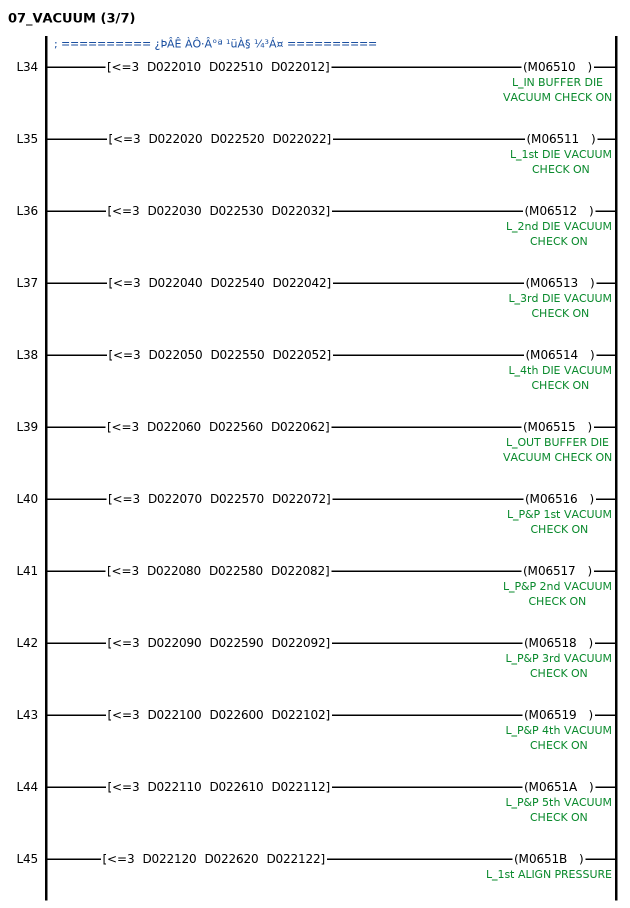
[picture p48: 07_VACUUM rungs L34-L45]
// ========== ¿ÞÂÊ ÀÔ·Â°ª ¹üÀ§ ¼³Á¤ ==========
; L34
LOAD<=3   D022010 D022510 D022012
OUT       M06510	// L_IN BUFFER DIE VACUUM CHECK ON
; L35
LOAD<=3   D022020 D022520 D022022
OUT       M06511	// L_1st DIE VACUUM CHECK ON
; L36
LOAD<=3   D022030 D022530 D022032
OUT       M06512	// L_2nd DIE VACUUM CHECK ON
; L37
LOAD<=3   D022040 D022540 D022042
OUT       M06513	// L_3rd DIE VACUUM CHECK ON
; L38
LOAD<=3   D022050 D022550 D022052
OUT       M06514	// L_4th DIE VACUUM CHECK ON
; L39
LOAD<=3   D022060 D022560 D022062
OUT       M06515	// L_OUT BUFFER DIE VACUUM CHECK ON
; L40
LOAD<=3   D022070 D022570 D022072
OUT       M06516	// L_P&P 1st VACUUM CHECK ON
; L41
LOAD<=3   D022080 D022580 D022082
OUT       M06517	// L_P&P 2nd VACUUM CHECK ON
; L42
LOAD<=3   D022090 D022590 D022092
OUT       M06518	// L_P&P 3rd VACUUM CHECK ON
; L43
LOAD<=3   D022100 D022600 D022102
OUT       M06519	// L_P&P 4th VACUUM CHECK ON
; L44
LOAD<=3   D022110 D022610 D022112
OUT       M0651A	// L_P&P 5th VACUUM CHECK ON
; L45
LOAD<=3   D022120 D022620 D022122
OUT       M0651B	// L_1st ALIGN PRESSURE

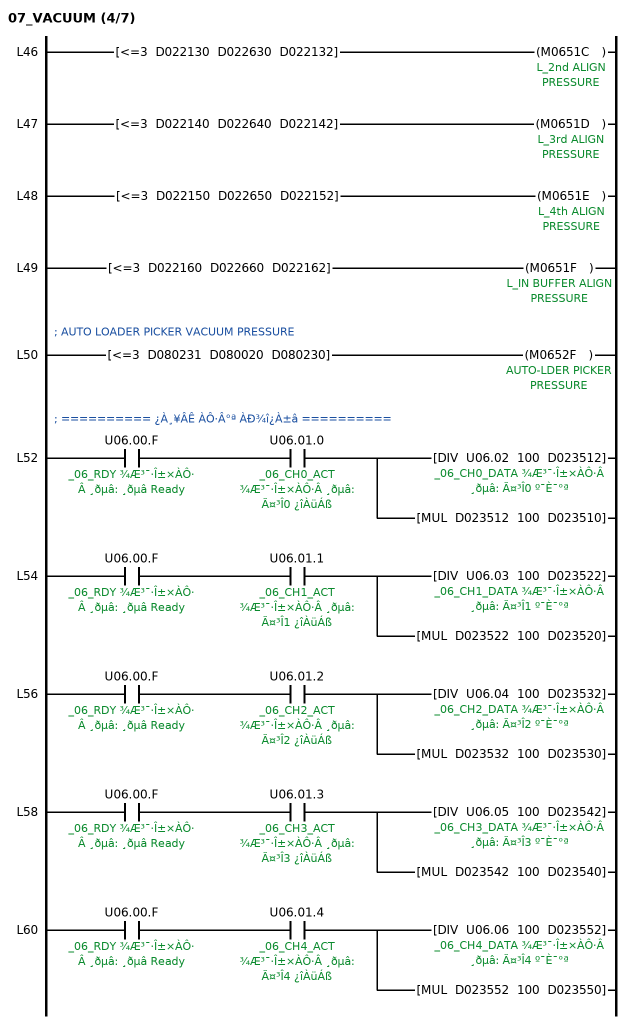
; L46
LOAD<=3   D022130 D022630 D022132
OUT       M0651C	// L_2nd ALIGN PRESSURE
; L47
LOAD<=3   D022140 D022640 D022142
OUT       M0651D	// L_3rd ALIGN PRESSURE
; L48
LOAD<=3   D022150 D022650 D022152
OUT       M0651E	// L_4th ALIGN PRESSURE
; L49
LOAD<=3   D022160 D022660 D022162
OUT       M0651F	// L_IN BUFFER ALIGN PRESSURE
; L50
LOAD<=3   D080231 D080020 D080230
OUT       M0652F	// AUTO-LDER PICKER PRESSURE
// output comment: AUTO LOADER PICKER VACUUM PRESSURE
// ========== ¿À¸¥ÂÊ ÀÔ·Â°ª ÀÐ¾î¿À±â ==========
; L52
LOAD      U06.00.F	// _06_RDY ¾Æ³¯·Î±×ÀÔ·Â ¸ðµâ: ¸ðµâ Ready
AND       U06.01.0	// _06_CH0_ACT ¾Æ³¯·Î±×ÀÔ·Â ¸ðµâ: Ã¤³Î0 ¿îÀüÁß
DIV       U06.02 100 D023512	// _06_CH0_DATA ¾Æ³¯·Î±×ÀÔ·Â ¸ðµâ: Ã¤³Î0 º¯È¯°ª
MUL       D023512 100 D023510
; L54
LOAD      U06.00.F	// _06_RDY ¾Æ³¯·Î±×ÀÔ·Â ¸ðµâ: ¸ðµâ Ready
AND       U06.01.1	// _06_CH1_ACT ¾Æ³¯·Î±×ÀÔ·Â ¸ðµâ: Ã¤³Î1 ¿îÀüÁß
DIV       U06.03 100 D023522	// _06_CH1_DATA ¾Æ³¯·Î±×ÀÔ·Â ¸ðµâ: Ã¤³Î1 º¯È¯°ª
MUL       D023522 100 D023520
; L56
LOAD      U06.00.F	// _06_RDY ¾Æ³¯·Î±×ÀÔ·Â ¸ðµâ: ¸ðµâ Ready
AND       U06.01.2	// _06_CH2_ACT ¾Æ³¯·Î±×ÀÔ·Â ¸ðµâ: Ã¤³Î2 ¿îÀüÁß
DIV       U06.04 100 D023532	// _06_CH2_DATA ¾Æ³¯·Î±×ÀÔ·Â ¸ðµâ: Ã¤³Î2 º¯È¯°ª
MUL       D023532 100 D023530
; L58
LOAD      U06.00.F	// _06_RDY ¾Æ³¯·Î±×ÀÔ·Â ¸ðµâ: ¸ðµâ Ready
AND       U06.01.3	// _06_CH3_ACT ¾Æ³¯·Î±×ÀÔ·Â ¸ðµâ: Ã¤³Î3 ¿îÀüÁß
DIV       U06.05 100 D023542	// _06_CH3_DATA ¾Æ³¯·Î±×ÀÔ·Â ¸ðµâ: Ã¤³Î3 º¯È¯°ª
MUL       D023542 100 D023540
; L60
LOAD      U06.00.F	// _06_RDY ¾Æ³¯·Î±×ÀÔ·Â ¸ðµâ: ¸ðµâ Ready
AND       U06.01.4	// _06_CH4_ACT ¾Æ³¯·Î±×ÀÔ·Â ¸ðµâ: Ã¤³Î4 ¿îÀüÁß
DIV       U06.06 100 D023552	// _06_CH4_DATA ¾Æ³¯·Î±×ÀÔ·Â ¸ðµâ: Ã¤³Î4 º¯È¯°ª
MUL       D023552 100 D023550

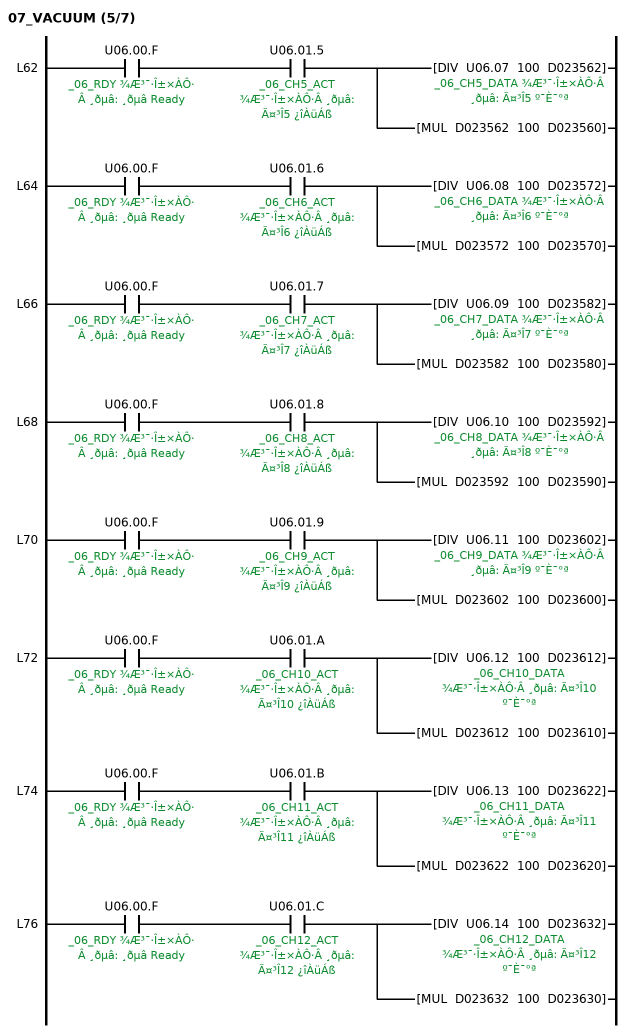
; L62
LOAD      U06.00.F	// _06_RDY ¾Æ³¯·Î±×ÀÔ·Â ¸ðµâ: ¸ðµâ Ready
AND       U06.01.5	// _06_CH5_ACT ¾Æ³¯·Î±×ÀÔ·Â ¸ðµâ: Ã¤³Î5 ¿îÀüÁß
DIV       U06.07 100 D023562	// _06_CH5_DATA ¾Æ³¯·Î±×ÀÔ·Â ¸ðµâ: Ã¤³Î5 º¯È¯°ª
MUL       D023562 100 D023560
; L64
LOAD      U06.00.F	// _06_RDY ¾Æ³¯·Î±×ÀÔ·Â ¸ðµâ: ¸ðµâ Ready
AND       U06.01.6	// _06_CH6_ACT ¾Æ³¯·Î±×ÀÔ·Â ¸ðµâ: Ã¤³Î6 ¿îÀüÁß
DIV       U06.08 100 D023572	// _06_CH6_DATA ¾Æ³¯·Î±×ÀÔ·Â ¸ðµâ: Ã¤³Î6 º¯È¯°ª
MUL       D023572 100 D023570
; L66
LOAD      U06.00.F	// _06_RDY ¾Æ³¯·Î±×ÀÔ·Â ¸ðµâ: ¸ðµâ Ready
AND       U06.01.7	// _06_CH7_ACT ¾Æ³¯·Î±×ÀÔ·Â ¸ðµâ: Ã¤³Î7 ¿îÀüÁß
DIV       U06.09 100 D023582	// _06_CH7_DATA ¾Æ³¯·Î±×ÀÔ·Â ¸ðµâ: Ã¤³Î7 º¯È¯°ª
MUL       D023582 100 D023580
; L68
LOAD      U06.00.F	// _06_RDY ¾Æ³¯·Î±×ÀÔ·Â ¸ðµâ: ¸ðµâ Ready
AND       U06.01.8	// _06_CH8_ACT ¾Æ³¯·Î±×ÀÔ·Â ¸ðµâ: Ã¤³Î8 ¿îÀüÁß
DIV       U06.10 100 D023592	// _06_CH8_DATA ¾Æ³¯·Î±×ÀÔ·Â ¸ðµâ: Ã¤³Î8 º¯È¯°ª
MUL       D023592 100 D023590
; L70
LOAD      U06.00.F	// _06_RDY ¾Æ³¯·Î±×ÀÔ·Â ¸ðµâ: ¸ðµâ Ready
AND       U06.01.9	// _06_CH9_ACT ¾Æ³¯·Î±×ÀÔ·Â ¸ðµâ: Ã¤³Î9 ¿îÀüÁß
DIV       U06.11 100 D023602	// _06_CH9_DATA ¾Æ³¯·Î±×ÀÔ·Â ¸ðµâ: Ã¤³Î9 º¯È¯°ª
MUL       D023602 100 D023600
; L72
LOAD      U06.00.F	// _06_RDY ¾Æ³¯·Î±×ÀÔ·Â ¸ðµâ: ¸ðµâ Ready
AND       U06.01.A	// _06_CH10_ACT ¾Æ³¯·Î±×ÀÔ·Â ¸ðµâ: Ã¤³Î10 ¿îÀüÁß
DIV       U06.12 100 D023612	// _06_CH10_DATA ¾Æ³¯·Î±×ÀÔ·Â ¸ðµâ: Ã¤³Î10 º¯È¯°ª
MUL       D023612 100 D023610
; L74
LOAD      U06.00.F	// _06_RDY ¾Æ³¯·Î±×ÀÔ·Â ¸ðµâ: ¸ðµâ Ready
AND       U06.01.B	// _06_CH11_ACT ¾Æ³¯·Î±×ÀÔ·Â ¸ðµâ: Ã¤³Î11 ¿îÀüÁß
DIV       U06.13 100 D023622	// _06_CH11_DATA ¾Æ³¯·Î±×ÀÔ·Â ¸ðµâ: Ã¤³Î11 º¯È¯°ª
MUL       D023622 100 D023620
; L76
LOAD      U06.00.F	// _06_RDY ¾Æ³¯·Î±×ÀÔ·Â ¸ðµâ: ¸ðµâ Ready
AND       U06.01.C	// _06_CH12_ACT ¾Æ³¯·Î±×ÀÔ·Â ¸ðµâ: Ã¤³Î12 ¿îÀüÁß
DIV       U06.14 100 D023632	// _06_CH12_DATA ¾Æ³¯·Î±×ÀÔ·Â ¸ðµâ: Ã¤³Î12 º¯È¯°ª
MUL       D023632 100 D023630

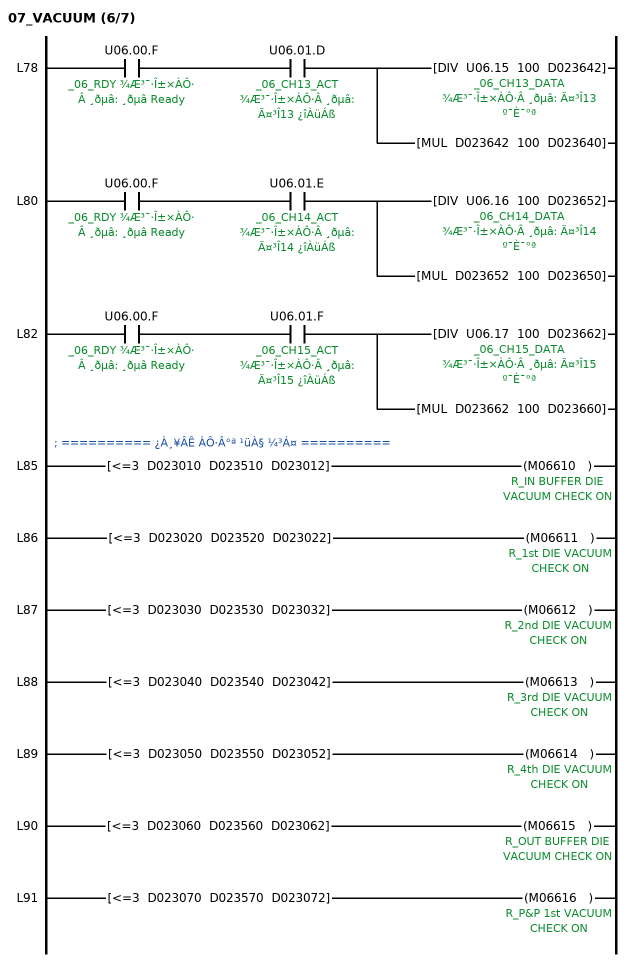
; L78
LOAD      U06.00.F	// _06_RDY ¾Æ³¯·Î±×ÀÔ·Â ¸ðµâ: ¸ðµâ Ready
AND       U06.01.D	// _06_CH13_ACT ¾Æ³¯·Î±×ÀÔ·Â ¸ðµâ: Ã¤³Î13 ¿îÀüÁß
DIV       U06.15 100 D023642	// _06_CH13_DATA ¾Æ³¯·Î±×ÀÔ·Â ¸ðµâ: Ã¤³Î13 º¯È¯°ª
MUL       D023642 100 D023640
; L80
LOAD      U06.00.F	// _06_RDY ¾Æ³¯·Î±×ÀÔ·Â ¸ðµâ: ¸ðµâ Ready
AND       U06.01.E	// _06_CH14_ACT ¾Æ³¯·Î±×ÀÔ·Â ¸ðµâ: Ã¤³Î14 ¿îÀüÁß
DIV       U06.16 100 D023652	// _06_CH14_DATA ¾Æ³¯·Î±×ÀÔ·Â ¸ðµâ: Ã¤³Î14 º¯È¯°ª
MUL       D023652 100 D023650
; L82
LOAD      U06.00.F	// _06_RDY ¾Æ³¯·Î±×ÀÔ·Â ¸ðµâ: ¸ðµâ Ready
AND       U06.01.F	// _06_CH15_ACT ¾Æ³¯·Î±×ÀÔ·Â ¸ðµâ: Ã¤³Î15 ¿îÀüÁß
DIV       U06.17 100 D023662	// _06_CH15_DATA ¾Æ³¯·Î±×ÀÔ·Â ¸ðµâ: Ã¤³Î15 º¯È¯°ª
MUL       D023662 100 D023660
// ========== ¿À¸¥ÂÊ ÀÔ·Â°ª ¹üÀ§ ¼³Á¤ ==========
; L85
LOAD<=3   D023010 D023510 D023012
OUT       M06610	// R_IN BUFFER DIE VACUUM CHECK ON
; L86
LOAD<=3   D023020 D023520 D023022
OUT       M06611	// R_1st DIE VACUUM CHECK ON
; L87
LOAD<=3   D023030 D023530 D023032
OUT       M06612	// R_2nd DIE VACUUM CHECK ON
; L88
LOAD<=3   D023040 D023540 D023042
OUT       M06613	// R_3rd DIE VACUUM CHECK ON
; L89
LOAD<=3   D023050 D023550 D023052
OUT       M06614	// R_4th DIE VACUUM CHECK ON
; L90
LOAD<=3   D023060 D023560 D023062
OUT       M06615	// R_OUT BUFFER DIE VACUUM CHECK ON
; L91
LOAD<=3   D023070 D023570 D023072
OUT       M06616	// R_P&P 1st VACUUM CHECK ON

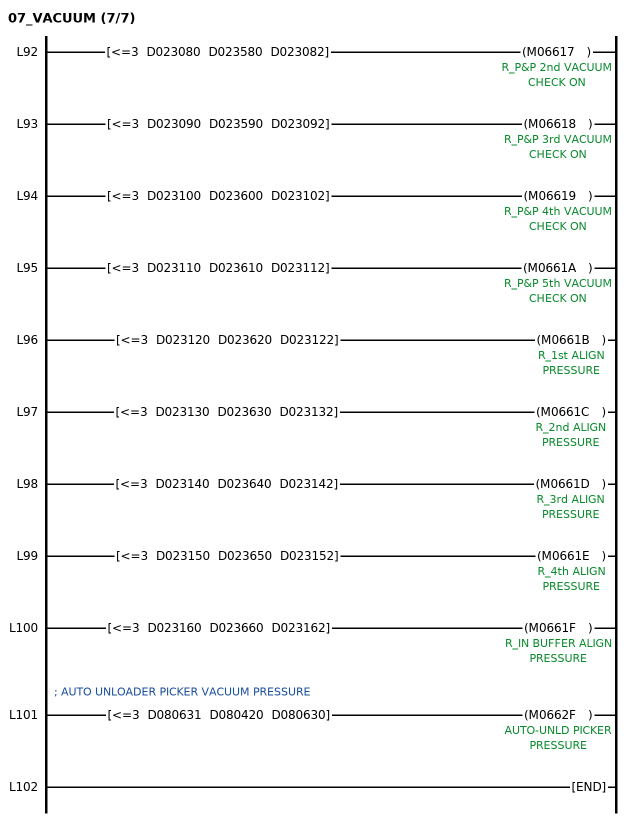
; L92
LOAD<=3   D023080 D023580 D023082
OUT       M06617	// R_P&P 2nd VACUUM CHECK ON
; L93
LOAD<=3   D023090 D023590 D023092
OUT       M06618	// R_P&P 3rd VACUUM CHECK ON
; L94
LOAD<=3   D023100 D023600 D023102
OUT       M06619	// R_P&P 4th VACUUM CHECK ON
; L95
LOAD<=3   D023110 D023610 D023112
OUT       M0661A	// R_P&P 5th VACUUM CHECK ON
; L96
LOAD<=3   D023120 D023620 D023122
OUT       M0661B	// R_1st ALIGN PRESSURE
; L97
LOAD<=3   D023130 D023630 D023132
OUT       M0661C	// R_2nd ALIGN PRESSURE
; L98
LOAD<=3   D023140 D023640 D023142
OUT       M0661D	// R_3rd ALIGN PRESSURE
; L99
LOAD<=3   D023150 D023650 D023152
OUT       M0661E	// R_4th ALIGN PRESSURE
; L100
LOAD<=3   D023160 D023660 D023162
OUT       M0661F	// R_IN BUFFER ALIGN PRESSURE
; L101
LOAD<=3   D080631 D080420 D080630
OUT       M0662F	// AUTO-UNLD PICKER PRESSURE
// output comment: AUTO UNLOADER PICKER VACUUM PRESSURE
; L102
END

PROGRAM 11_L_1st_MAND (task: ½ºÄµ ÇÁ·Î±×·¥)

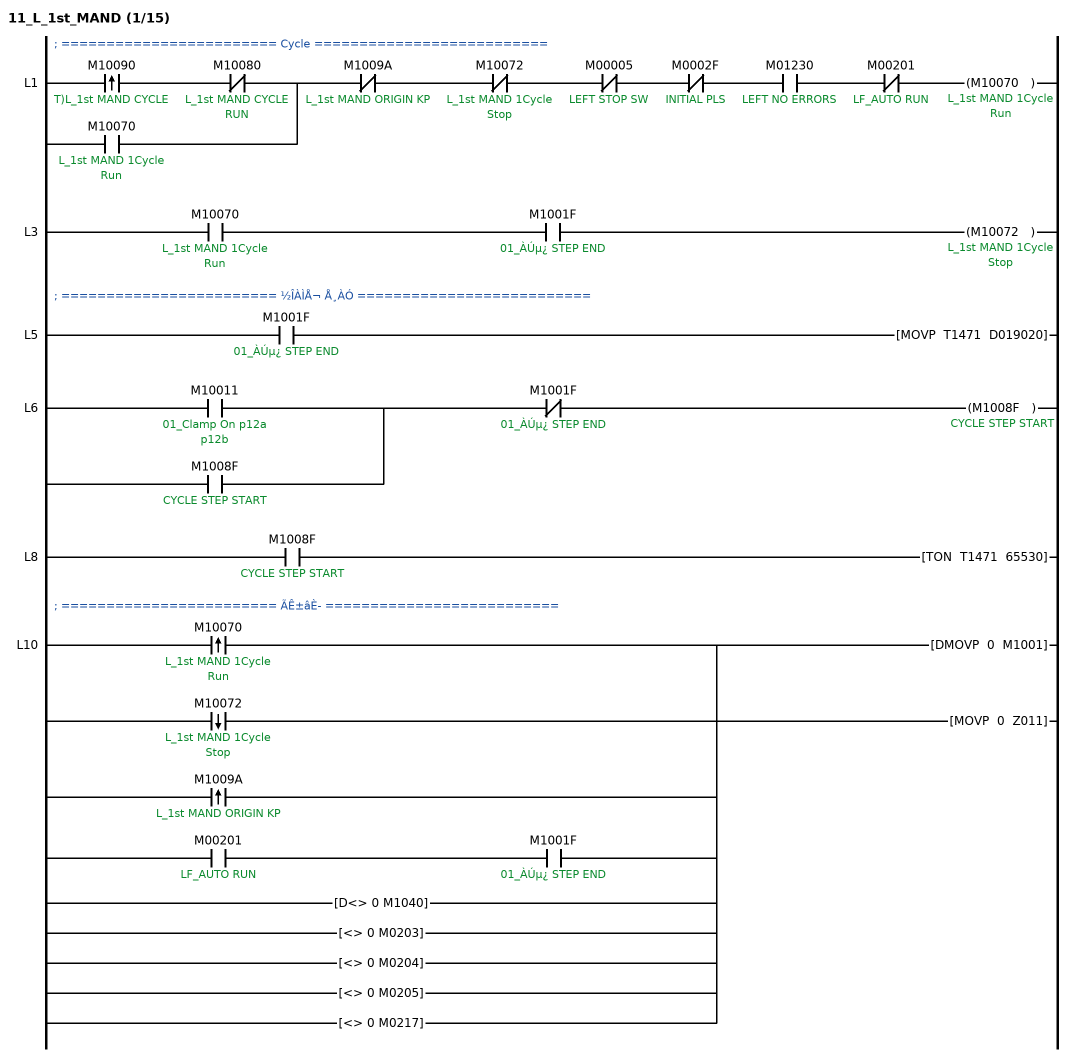
// ======================== Cycle ==========================
; L1
LOADP     M10090	// T)L_1st MAND CYCLE
AND NOT   M10080	// L_1st MAND CYCLE RUN
OR        M10070	// L_1st MAND 1Cycle Run
AND NOT   M1009A	// L_1st MAND ORIGIN KP
AND NOT   M10072	// L_1st MAND 1Cycle Stop
AND NOT   M00005	// LEFT STOP SW
AND NOT   M0002F	// INITIAL PLS
AND       M01230	// LEFT NO ERRORS
AND NOT   M00201	// LF_AUTO RUN
OUT       M10070	// L_1st MAND 1Cycle Run
; L3
LOAD      M10070	// L_1st MAND 1Cycle Run
AND       M1001F	// 01_ÀÚµ¿ STEP END
OUT       M10072	// L_1st MAND 1Cycle Stop
// ======================== ½ÎÀÌÅ¬ Å¸ÀÓ ==========================
; L5
LOAD      M1001F	// 01_ÀÚµ¿ STEP END
MOVP      T1471 D019020
; L6
LOAD      M10011	// 01_Clamp On p12a p12b
OR        M1008F	// CYCLE STEP START
AND NOT   M1001F	// 01_ÀÚµ¿ STEP END
OUT       M1008F	// CYCLE STEP START
; L8
LOAD      M1008F	// CYCLE STEP START
TON       T1471 65530
// ======================== ÃÊ±âÈ­ ==========================
; L10
LOADP     M10070	// L_1st MAND 1Cycle Run
ORN       M10072	// L_1st MAND 1Cycle Stop
ORP       M1009A	// L_1st MAND ORIGIN KP
LOAD      M00201	// LF_AUTO RUN
AND       M1001F	// 01_ÀÚµ¿ STEP END
OR LOAD
ORD<>     0 M1040
OR<>      0 M0203
OR<>      0 M0204
OR<>      0 M0205
OR<>      0 M0217
DMOVP     0 M1001
MOVP      0 Z011

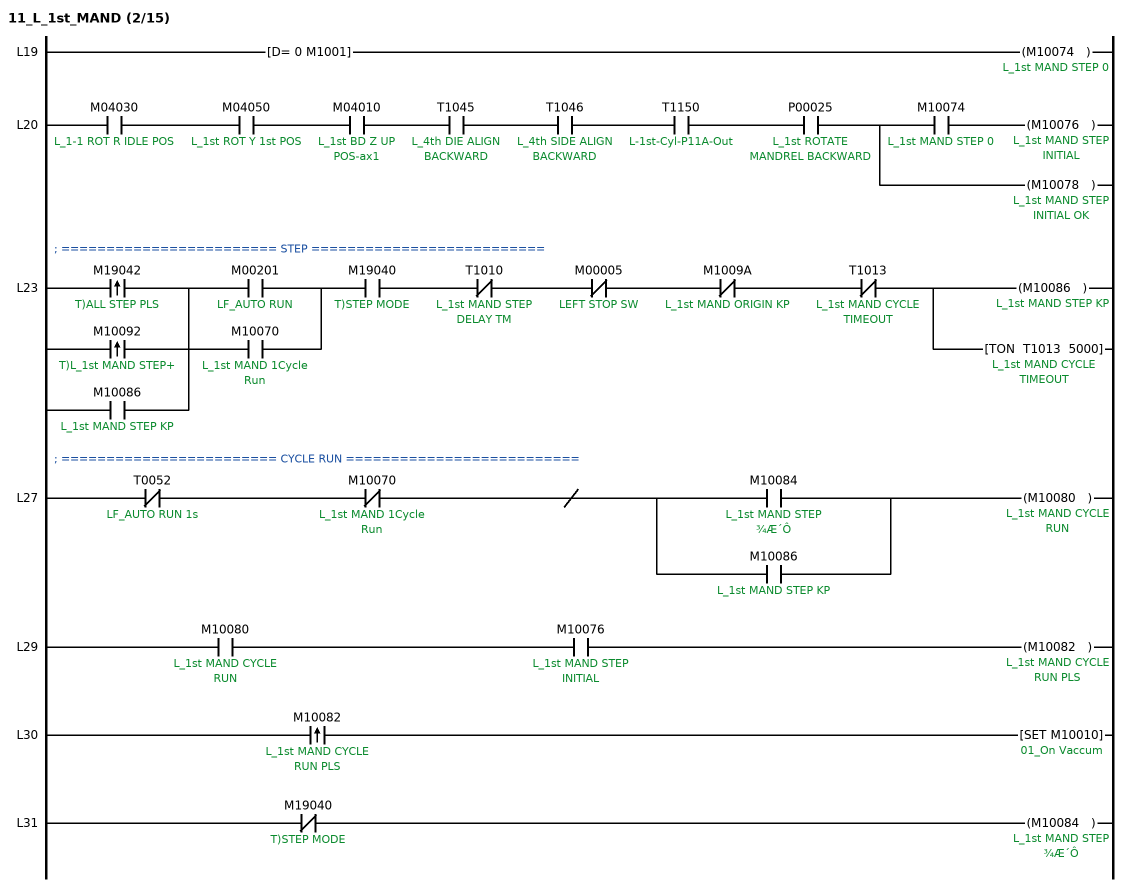
; L19
LOADD=    0 M1001
OUT       M10074	// L_1st MAND STEP 0
; L20
LOAD      M04030	// L_1-1 ROT R IDLE POS
AND       M04050	// L_1st ROT Y 1st POS
AND       M04010	// L_1st BD Z UP POS-ax1
AND       T1045	// L_4th DIE ALIGN BACKWARD
AND       T1046	// L_4th SIDE ALIGN BACKWARD
AND       T1150	// L-1st-Cyl-P11A-Out
AND       P00025	// L_1st ROTATE MANDREL BACKWARD
MPUSH
AND       M10074	// L_1st MAND STEP 0
OUT       M10076	// L_1st MAND STEP INITIAL
MPOP
OUT       M10078	// L_1st MAND STEP INITIAL OK
// ======================== STEP ==========================
; L23
LOADP     M19042	// T)ALL STEP PLS
ORP       M10092	// T)L_1st MAND STEP+
OR        M10086	// L_1st MAND STEP KP
LOAD      M00201	// LF_AUTO RUN
OR        M10070	// L_1st MAND 1Cycle Run
AND LOAD
AND       M19040	// T)STEP MODE
AND NOT   T1010	// L_1st MAND STEP DELAY TM
AND NOT   M00005	// LEFT STOP SW
AND NOT   M1009A	// L_1st MAND ORIGIN KP
AND NOT   T1013	// L_1st MAND CYCLE TIMEOUT
OUT       M10086	// L_1st MAND STEP KP
TON       T1013 5000	// L_1st MAND CYCLE TIMEOUT
// ======================== CYCLE RUN ==========================
; L27
LOAD NOT  T0052	// LF_AUTO RUN 1s
AND NOT   M10070	// L_1st MAND 1Cycle Run
NOT
LOAD      M10084	// L_1st MAND STEP ¾Æ´Ô
OR        M10086	// L_1st MAND STEP KP
AND LOAD
OUT       M10080	// L_1st MAND CYCLE RUN
; L29
LOAD      M10080	// L_1st MAND CYCLE RUN
AND       M10076	// L_1st MAND STEP INITIAL
OUT       M10082	// L_1st MAND CYCLE RUN PLS
; L30
LOADP     M10082	// L_1st MAND CYCLE RUN PLS
SET       M10010	// 01_On Vaccum
; L31
LOAD NOT  M19040	// T)STEP MODE
OUT       M10084	// L_1st MAND STEP ¾Æ´Ô

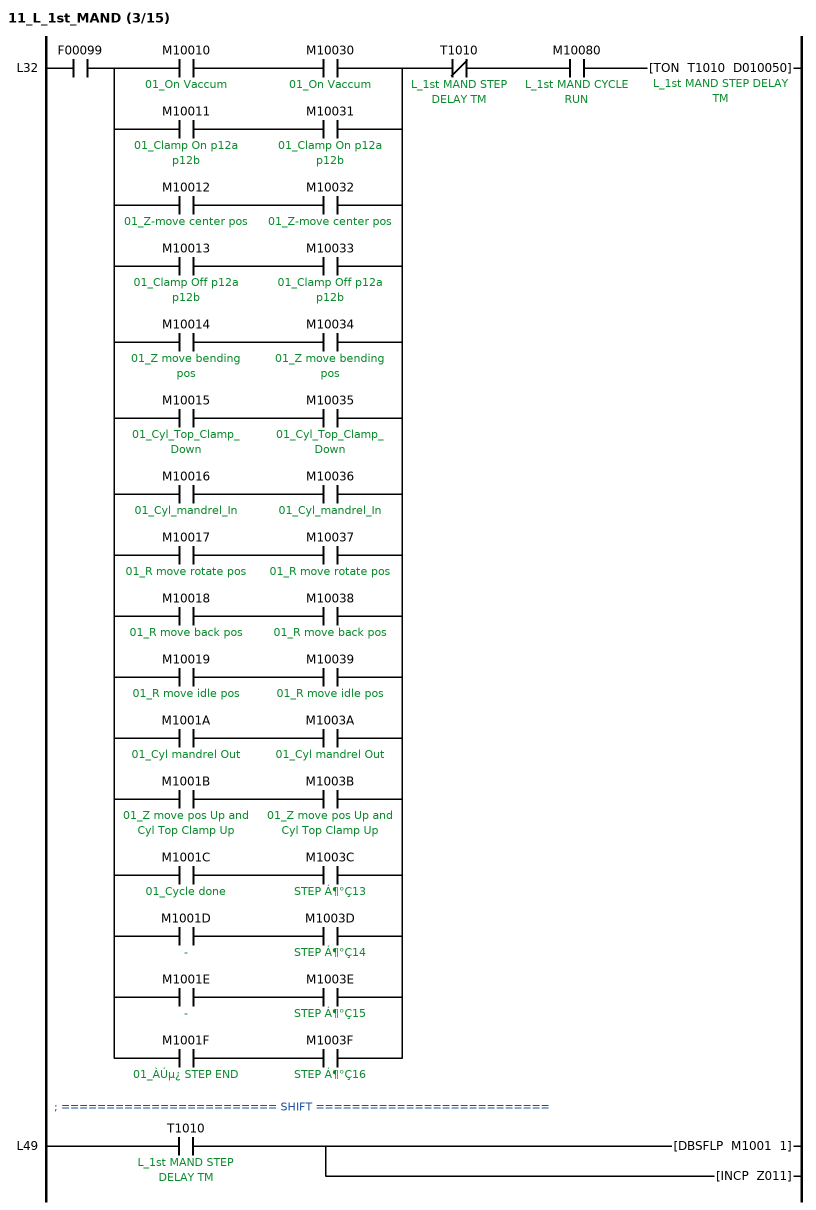
; L32
LOAD      F00099
LOAD      M10010	// 01_On Vaccum
AND       M10030	// 01_On Vaccum
LOAD      M10011	// 01_Clamp On p12a p12b
AND       M10031	// 01_Clamp On p12a p12b
OR LOAD
LOAD      M10012	// 01_Z-move center pos
AND       M10032	// 01_Z-move center pos
OR LOAD
LOAD      M10013	// 01_Clamp Off p12a p12b
AND       M10033	// 01_Clamp Off p12a p12b
OR LOAD
LOAD      M10014	// 01_Z move bending pos
AND       M10034	// 01_Z move bending pos
OR LOAD
LOAD      M10015	// 01_Cyl_Top_Clamp_Down
AND       M10035	// 01_Cyl_Top_Clamp_Down
OR LOAD
LOAD      M10016	// 01_Cyl_mandrel_In
AND       M10036	// 01_Cyl_mandrel_In
OR LOAD
LOAD      M10017	// 01_R move rotate pos
AND       M10037	// 01_R move rotate pos
OR LOAD
LOAD      M10018	// 01_R move back pos
AND       M10038	// 01_R move back pos
OR LOAD
LOAD      M10019	// 01_R move idle pos
AND       M10039	// 01_R move idle pos
OR LOAD
LOAD      M1001A	// 01_Cyl mandrel Out
AND       M1003A	// 01_Cyl mandrel Out
OR LOAD
LOAD      M1001B	// 01_Z move pos Up and Cyl Top Clamp Up
AND       M1003B	// 01_Z move pos Up and Cyl Top Clamp Up
OR LOAD
LOAD      M1001C	// 01_Cycle done
AND       M1003C	// STEP Á¶°Ç13
OR LOAD
LOAD      M1001D	// -
AND       M1003D	// STEP Á¶°Ç14
OR LOAD
LOAD      M1001E	// -
AND       M1003E	// STEP Á¶°Ç15
OR LOAD
LOAD      M1001F	// 01_ÀÚµ¿ STEP END
AND       M1003F	// STEP Á¶°Ç16
OR LOAD
AND LOAD
AND NOT   T1010	// L_1st MAND STEP DELAY TM
AND       M10080	// L_1st MAND CYCLE RUN
TON       T1010 D010050	// L_1st MAND STEP DELAY TM
// ======================== SHIFT ==========================
; L49
LOAD      T1010	// L_1st MAND STEP DELAY TM
DBSFLP    M1001 1
INCP      Z011

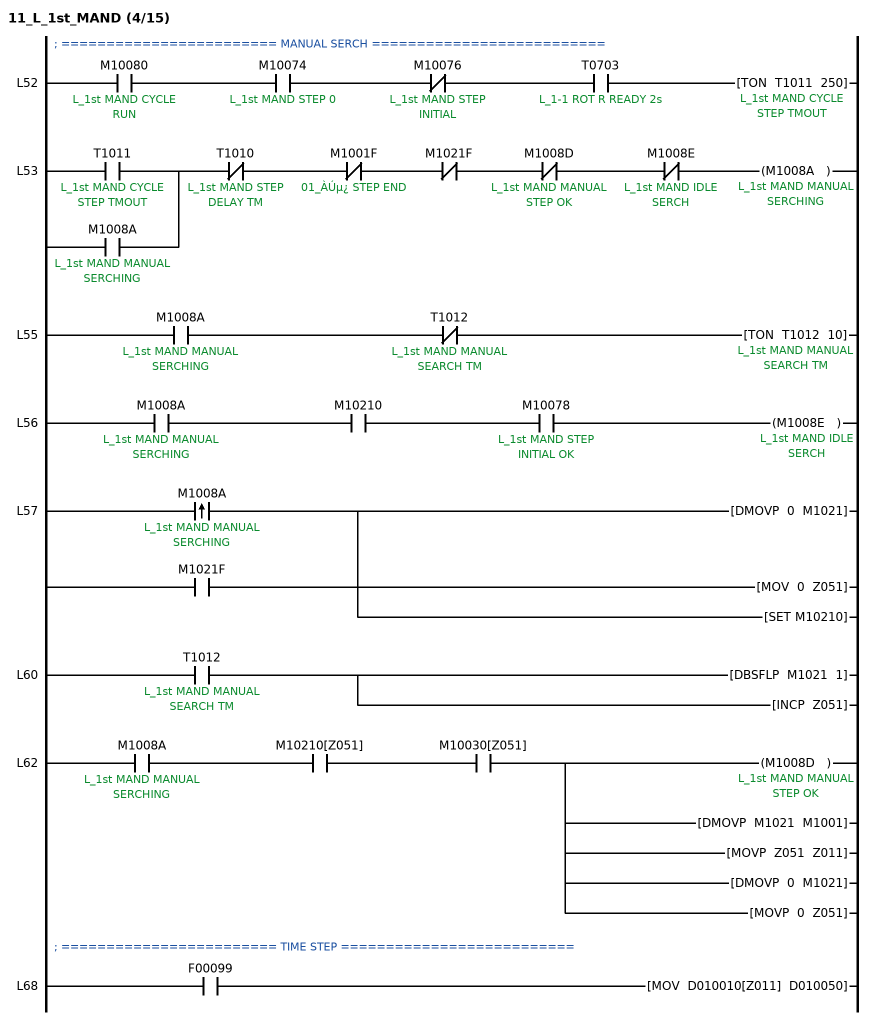
// ======================== MANUAL SERCH ==========================
; L52
LOAD      M10080	// L_1st MAND CYCLE RUN
AND       M10074	// L_1st MAND STEP 0
AND NOT   M10076	// L_1st MAND STEP INITIAL
AND       T0703	// L_1-1 ROT R READY 2s
TON       T1011 250	// L_1st MAND CYCLE STEP TMOUT
; L53
LOAD      T1011	// L_1st MAND CYCLE STEP TMOUT
OR        M1008A	// L_1st MAND MANUAL SERCHING
AND NOT   T1010	// L_1st MAND STEP DELAY TM
AND NOT   M1001F	// 01_ÀÚµ¿ STEP END
AND NOT   M1021F
AND NOT   M1008D	// L_1st MAND MANUAL STEP OK
AND NOT   M1008E	// L_1st MAND IDLE SERCH
OUT       M1008A	// L_1st MAND MANUAL SERCHING
; L55
LOAD      M1008A	// L_1st MAND MANUAL SERCHING
AND NOT   T1012	// L_1st MAND MANUAL SEARCH TM
TON       T1012 10	// L_1st MAND MANUAL SEARCH TM
; L56
LOAD      M1008A	// L_1st MAND MANUAL SERCHING
AND       M10210
AND       M10078	// L_1st MAND STEP INITIAL OK
OUT       M1008E	// L_1st MAND IDLE SERCH
; L57
LOADP     M1008A	// L_1st MAND MANUAL SERCHING
OR        M1021F
DMOVP     0 M1021
MOV       0 Z051
SET       M10210
; L60
LOAD      T1012	// L_1st MAND MANUAL SEARCH TM
DBSFLP    M1021 1
INCP      Z051
; L62
LOAD      M1008A	// L_1st MAND MANUAL SERCHING
AND       M10210[Z051]
AND       M10030[Z051]
OUT       M1008D	// L_1st MAND MANUAL STEP OK
DMOVP     M1021 M1001
MOVP      Z051 Z011
DMOVP     0 M1021
MOVP      0 Z051
// ======================== TIME STEP ==========================
; L68
LOAD      F00099
MOV       D010010[Z011] D010050

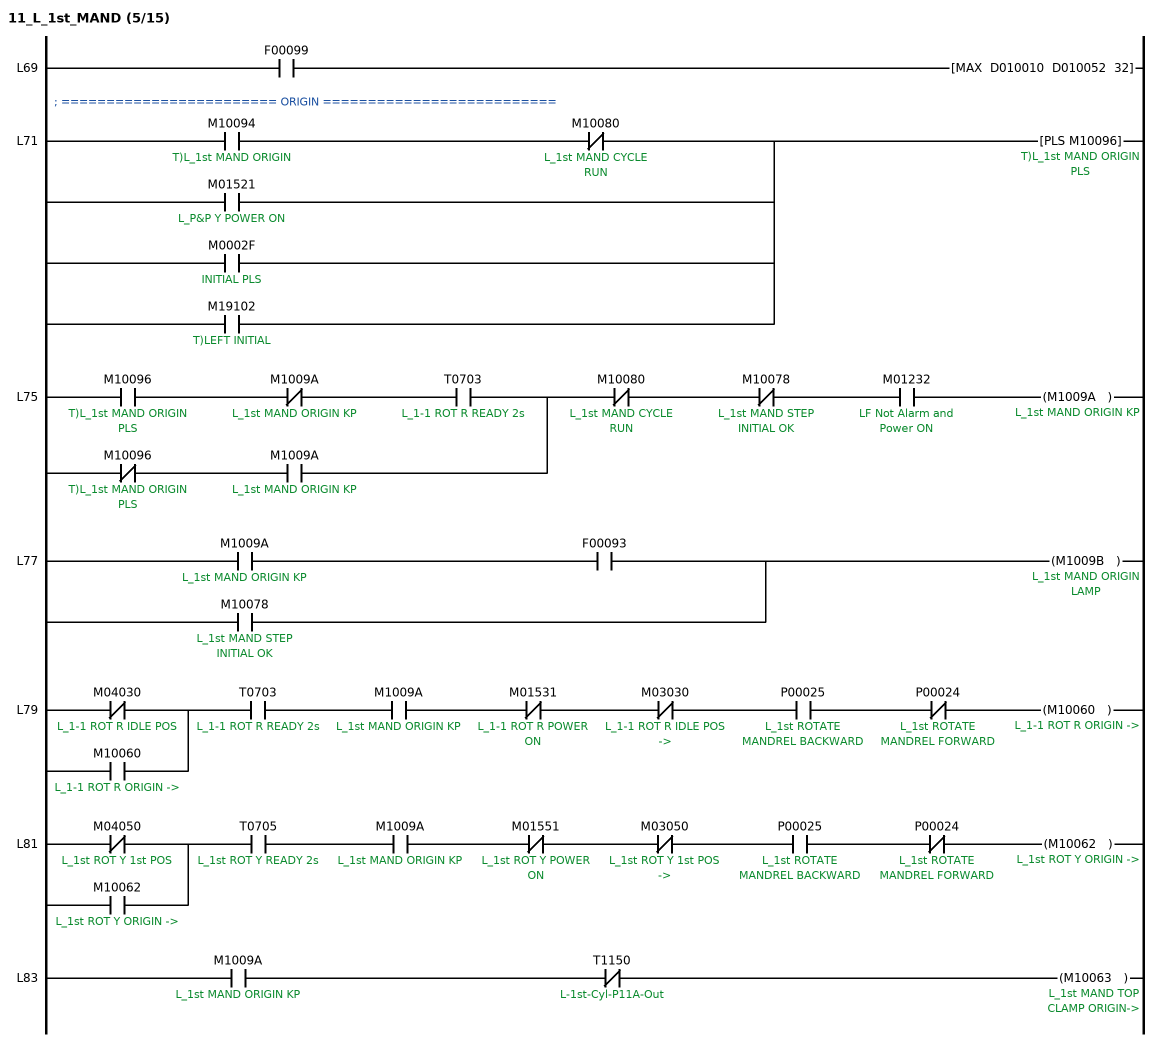
; L69
LOAD      F00099
MAX       D010010 D010052 32
// ======================== ORIGIN ==========================
; L71
LOAD      M10094	// T)L_1st MAND ORIGIN
AND NOT   M10080	// L_1st MAND CYCLE RUN
OR        M01521	// L_P&P Y POWER ON
OR        M0002F	// INITIAL PLS
OR        M19102	// T)LEFT INITIAL
OUTP      M10096	// T)L_1st MAND ORIGIN PLS
; L75
LOAD      M10096	// T)L_1st MAND ORIGIN PLS
AND NOT   M1009A	// L_1st MAND ORIGIN KP
AND       T0703	// L_1-1 ROT R READY 2s
LOAD NOT  M10096	// T)L_1st MAND ORIGIN PLS
AND       M1009A	// L_1st MAND ORIGIN KP
OR LOAD
AND NOT   M10080	// L_1st MAND CYCLE RUN
AND NOT   M10078	// L_1st MAND STEP INITIAL OK
AND       M01232	// LF Not Alarm and Power ON
OUT       M1009A	// L_1st MAND ORIGIN KP
; L77
LOAD      M1009A	// L_1st MAND ORIGIN KP
AND       F00093
OR        M10078	// L_1st MAND STEP INITIAL OK
OUT       M1009B	// L_1st MAND ORIGIN LAMP
; L79
LOAD NOT  M04030	// L_1-1 ROT R IDLE POS
OR        M10060	// L_1-1 ROT R ORIGIN ->
AND       T0703	// L_1-1 ROT R READY 2s
AND       M1009A	// L_1st MAND ORIGIN KP
AND NOT   M01531	// L_1-1 ROT R POWER ON
AND NOT   M03030	// L_1-1 ROT R IDLE POS ->
AND       P00025	// L_1st ROTATE MANDREL BACKWARD
AND NOT   P00024	// L_1st ROTATE MANDREL FORWARD
OUT       M10060	// L_1-1 ROT R ORIGIN ->
; L81
LOAD NOT  M04050	// L_1st ROT Y 1st POS
OR        M10062	// L_1st ROT Y ORIGIN ->
AND       T0705	// L_1st ROT Y READY 2s
AND       M1009A	// L_1st MAND ORIGIN KP
AND NOT   M01551	// L_1st ROT Y POWER ON
AND NOT   M03050	// L_1st ROT Y 1st POS ->
AND       P00025	// L_1st ROTATE MANDREL BACKWARD
AND NOT   P00024	// L_1st ROTATE MANDREL FORWARD
OUT       M10062	// L_1st ROT Y ORIGIN ->
; L83
LOAD      M1009A	// L_1st MAND ORIGIN KP
AND NOT   T1150	// L-1st-Cyl-P11A-Out
OUT       M10063	// L_1st MAND TOP CLAMP ORIGIN->

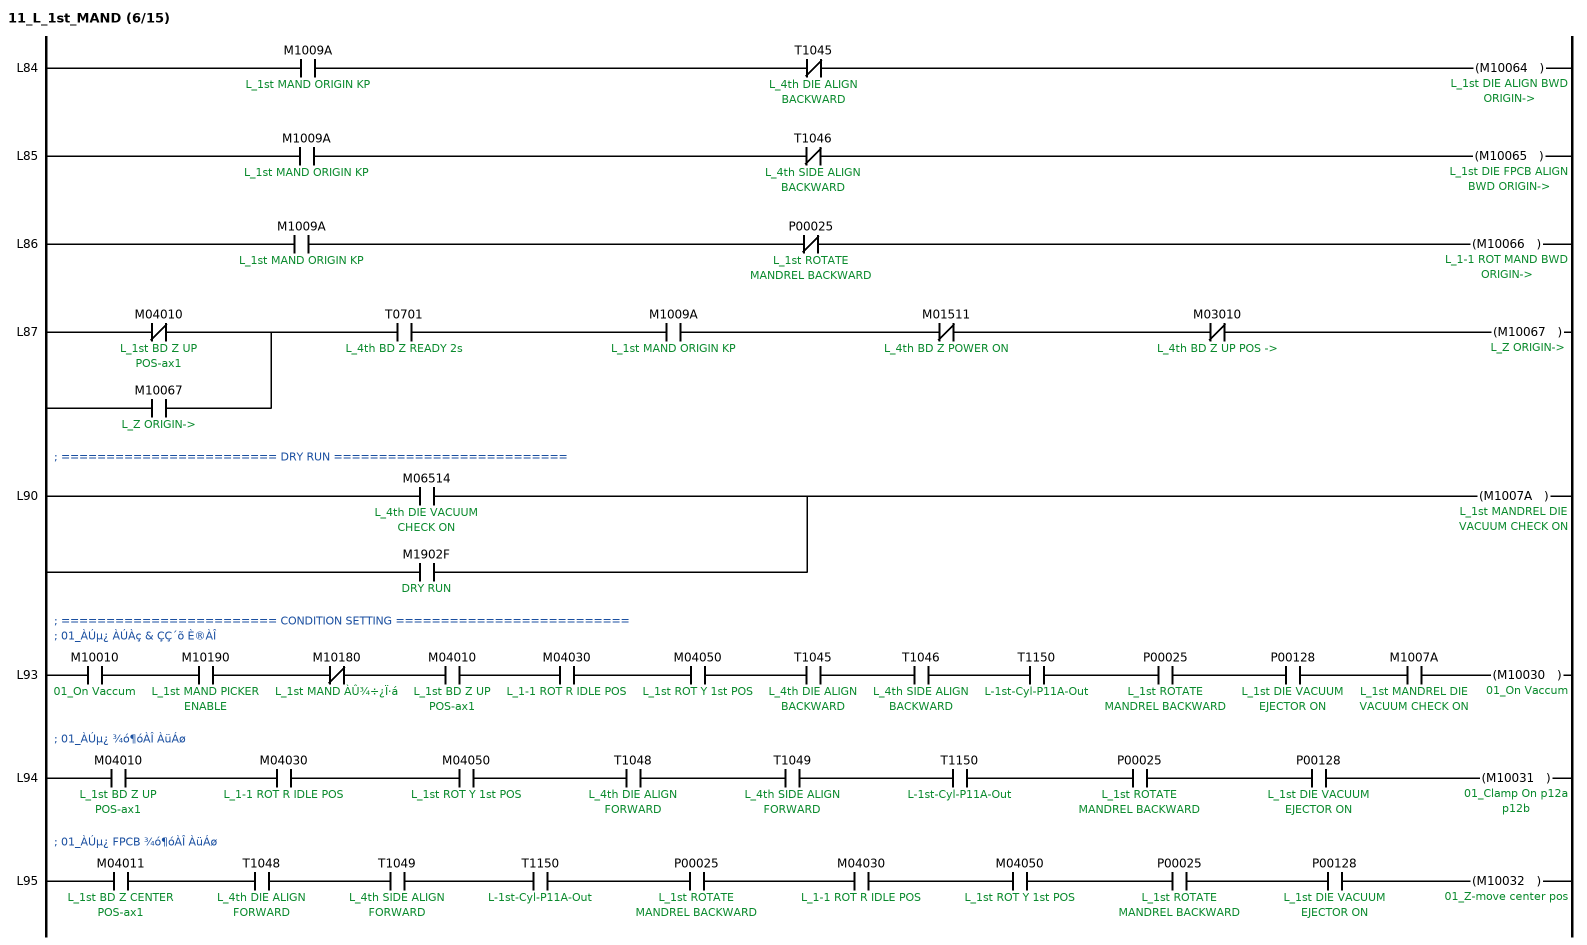
; L84
LOAD      M1009A	// L_1st MAND ORIGIN KP
AND NOT   T1045	// L_4th DIE ALIGN BACKWARD
OUT       M10064	// L_1st DIE ALIGN BWD ORIGIN->
; L85
LOAD      M1009A	// L_1st MAND ORIGIN KP
AND NOT   T1046	// L_4th SIDE ALIGN BACKWARD
OUT       M10065	// L_1st DIE FPCB ALIGN BWD ORIGIN->
; L86
LOAD      M1009A	// L_1st MAND ORIGIN KP
AND NOT   P00025	// L_1st ROTATE MANDREL BACKWARD
OUT       M10066	// L_1-1 ROT MAND BWD ORIGIN->
; L87
LOAD NOT  M04010	// L_1st BD Z UP POS-ax1
OR        M10067	// L_Z ORIGIN->
AND       T0701	// L_4th BD Z READY 2s
AND       M1009A	// L_1st MAND ORIGIN KP
AND NOT   M01511	// L_4th BD Z POWER ON
AND NOT   M03010	// L_4th BD Z UP POS ->
OUT       M10067	// L_Z ORIGIN->
// ======================== DRY RUN ==========================
; L90
LOAD      M06514	// L_4th DIE VACUUM CHECK ON
OR        M1902F	// DRY RUN
OUT       M1007A	// L_1st MANDREL DIE VACUUM CHECK ON
// ======================== CONDITION SETTING ==========================
; L93
LOAD      M10010	// 01_On Vaccum
AND       M10190	// L_1st MAND PICKER ENABLE
AND NOT   M10180	// L_1st MAND ÀÛ¾÷¿Ï·á
AND       M04010	// L_1st BD Z UP POS-ax1
AND       M04030	// L_1-1 ROT R IDLE POS
AND       M04050	// L_1st ROT Y 1st POS
AND       T1045	// L_4th DIE ALIGN BACKWARD
AND       T1046	// L_4th SIDE ALIGN BACKWARD
AND       T1150	// L-1st-Cyl-P11A-Out
AND       P00025	// L_1st ROTATE MANDREL BACKWARD
AND       P00128	// L_1st DIE VACUUM EJECTOR ON
AND       M1007A	// L_1st MANDREL DIE VACUUM CHECK ON
OUT       M10030	// 01_On Vaccum
// output comment: 01_ÀÚµ¿ ÀÚÀç & ÇÇ´õ È®ÀÎ
; L94
LOAD      M04010	// L_1st BD Z UP POS-ax1
AND       M04030	// L_1-1 ROT R IDLE POS
AND       M04050	// L_1st ROT Y 1st POS
AND       T1048	// L_4th DIE ALIGN FORWARD
AND       T1049	// L_4th SIDE ALIGN FORWARD
AND       T1150	// L-1st-Cyl-P11A-Out
AND       P00025	// L_1st ROTATE MANDREL BACKWARD
AND       P00128	// L_1st DIE VACUUM EJECTOR ON
OUT       M10031	// 01_Clamp On p12a p12b
// output comment: 01_ÀÚµ¿ ¾ó¶óÀÎ ÀüÁø
; L95
LOAD      M04011	// L_1st BD Z CENTER POS-ax1
AND       T1048	// L_4th DIE ALIGN FORWARD
AND       T1049	// L_4th SIDE ALIGN FORWARD
AND       T1150	// L-1st-Cyl-P11A-Out
AND       P00025	// L_1st ROTATE MANDREL BACKWARD
AND       M04030	// L_1-1 ROT R IDLE POS
AND       M04050	// L_1st ROT Y 1st POS
AND       P00025	// L_1st ROTATE MANDREL BACKWARD
AND       P00128	// L_1st DIE VACUUM EJECTOR ON
OUT       M10032	// 01_Z-move center pos
// output comment: 01_ÀÚµ¿ FPCB ¾ó¶óÀÎ ÀüÁø

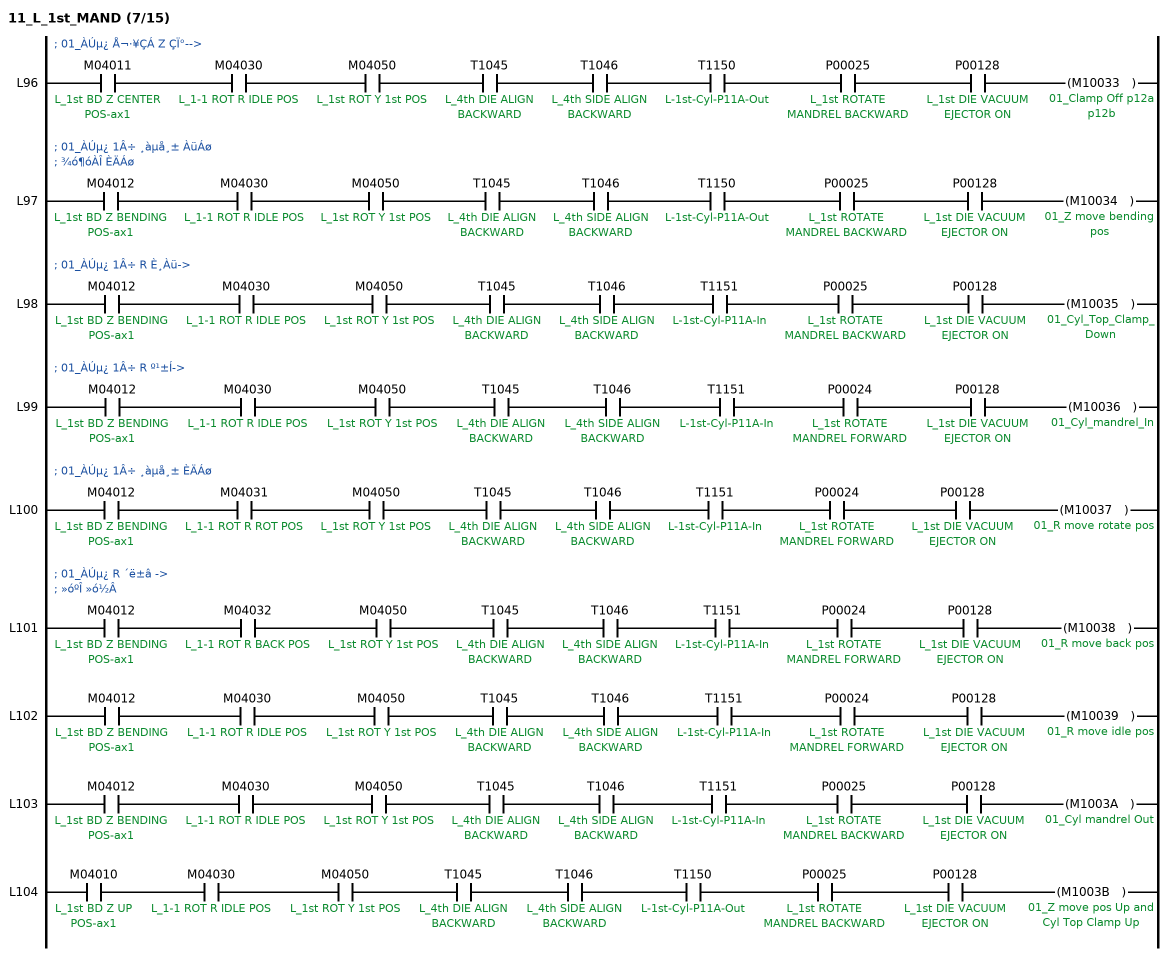
; L96
LOAD      M04011	// L_1st BD Z CENTER POS-ax1
AND       M04030	// L_1-1 ROT R IDLE POS
AND       M04050	// L_1st ROT Y 1st POS
AND       T1045	// L_4th DIE ALIGN BACKWARD
AND       T1046	// L_4th SIDE ALIGN BACKWARD
AND       T1150	// L-1st-Cyl-P11A-Out
AND       P00025	// L_1st ROTATE MANDREL BACKWARD
AND       P00128	// L_1st DIE VACUUM EJECTOR ON
OUT       M10033	// 01_Clamp Off p12a p12b
// output comment: 01_ÀÚµ¿ Å¬·¥ÇÁ Z ÇÏ°­->
; L97
LOAD      M04012	// L_1st BD Z BENDING POS-ax1
AND       M04030	// L_1-1 ROT R IDLE POS
AND       M04050	// L_1st ROT Y 1st POS
AND       T1045	// L_4th DIE ALIGN BACKWARD
AND       T1046	// L_4th SIDE ALIGN BACKWARD
AND       T1150	// L-1st-Cyl-P11A-Out
AND       P00025	// L_1st ROTATE MANDREL BACKWARD
AND       P00128	// L_1st DIE VACUUM EJECTOR ON
OUT       M10034	// 01_Z move bending pos
// output comment: 01_ÀÚµ¿ 1Â÷ ¸àµå¸± ÀüÁø ¾ó¶óÀÎ ÈÄÁø
; L98
LOAD      M04012	// L_1st BD Z BENDING POS-ax1
AND       M04030	// L_1-1 ROT R IDLE POS
AND       M04050	// L_1st ROT Y 1st POS
AND       T1045	// L_4th DIE ALIGN BACKWARD
AND       T1046	// L_4th SIDE ALIGN BACKWARD
AND       T1151	// L-1st-Cyl-P11A-In
AND       P00025	// L_1st ROTATE MANDREL BACKWARD
AND       P00128	// L_1st DIE VACUUM EJECTOR ON
OUT       M10035	// 01_Cyl_Top_Clamp_Down
// output comment: 01_ÀÚµ¿ 1Â÷ R È¸Àü->
; L99
LOAD      M04012	// L_1st BD Z BENDING POS-ax1
AND       M04030	// L_1-1 ROT R IDLE POS
AND       M04050	// L_1st ROT Y 1st POS
AND       T1045	// L_4th DIE ALIGN BACKWARD
AND       T1046	// L_4th SIDE ALIGN BACKWARD
AND       T1151	// L-1st-Cyl-P11A-In
AND       P00024	// L_1st ROTATE MANDREL FORWARD
AND       P00128	// L_1st DIE VACUUM EJECTOR ON
OUT       M10036	// 01_Cyl_mandrel_In
// output comment: 01_ÀÚµ¿ 1Â÷ R º¹±Í->
; L100
LOAD      M04012	// L_1st BD Z BENDING POS-ax1
AND       M04031	// L_1-1 ROT R ROT POS
AND       M04050	// L_1st ROT Y 1st POS
AND       T1045	// L_4th DIE ALIGN BACKWARD
AND       T1046	// L_4th SIDE ALIGN BACKWARD
AND       T1151	// L-1st-Cyl-P11A-In
AND       P00024	// L_1st ROTATE MANDREL FORWARD
AND       P00128	// L_1st DIE VACUUM EJECTOR ON
OUT       M10037	// 01_R move rotate pos
// output comment: 01_ÀÚµ¿ 1Â÷ ¸àµå¸± ÈÄÁø
; L101
LOAD      M04012	// L_1st BD Z BENDING POS-ax1
AND       M04032	// L_1-1 ROT R BACK POS
AND       M04050	// L_1st ROT Y 1st POS
AND       T1045	// L_4th DIE ALIGN BACKWARD
AND       T1046	// L_4th SIDE ALIGN BACKWARD
AND       T1151	// L-1st-Cyl-P11A-In
AND       P00024	// L_1st ROTATE MANDREL FORWARD
AND       P00128	// L_1st DIE VACUUM EJECTOR ON
OUT       M10038	// 01_R move back pos
// output comment: 01_ÀÚµ¿ R ´ë±â -> »óºÎ »ó½Â
; L102
LOAD      M04012	// L_1st BD Z BENDING POS-ax1
AND       M04030	// L_1-1 ROT R IDLE POS
AND       M04050	// L_1st ROT Y 1st POS
AND       T1045	// L_4th DIE ALIGN BACKWARD
AND       T1046	// L_4th SIDE ALIGN BACKWARD
AND       T1151	// L-1st-Cyl-P11A-In
AND       P00024	// L_1st ROTATE MANDREL FORWARD
AND       P00128	// L_1st DIE VACUUM EJECTOR ON
OUT       M10039	// 01_R move idle pos
; L103
LOAD      M04012	// L_1st BD Z BENDING POS-ax1
AND       M04030	// L_1-1 ROT R IDLE POS
AND       M04050	// L_1st ROT Y 1st POS
AND       T1045	// L_4th DIE ALIGN BACKWARD
AND       T1046	// L_4th SIDE ALIGN BACKWARD
AND       T1151	// L-1st-Cyl-P11A-In
AND       P00025	// L_1st ROTATE MANDREL BACKWARD
AND       P00128	// L_1st DIE VACUUM EJECTOR ON
OUT       M1003A	// 01_Cyl mandrel Out
; L104
LOAD      M04010	// L_1st BD Z UP POS-ax1
AND       M04030	// L_1-1 ROT R IDLE POS
AND       M04050	// L_1st ROT Y 1st POS
AND       T1045	// L_4th DIE ALIGN BACKWARD
AND       T1046	// L_4th SIDE ALIGN BACKWARD
AND       T1150	// L-1st-Cyl-P11A-Out
AND       P00025	// L_1st ROTATE MANDREL BACKWARD
AND       P00128	// L_1st DIE VACUUM EJECTOR ON
OUT       M1003B	// 01_Z move pos Up and Cyl Top Clamp Up

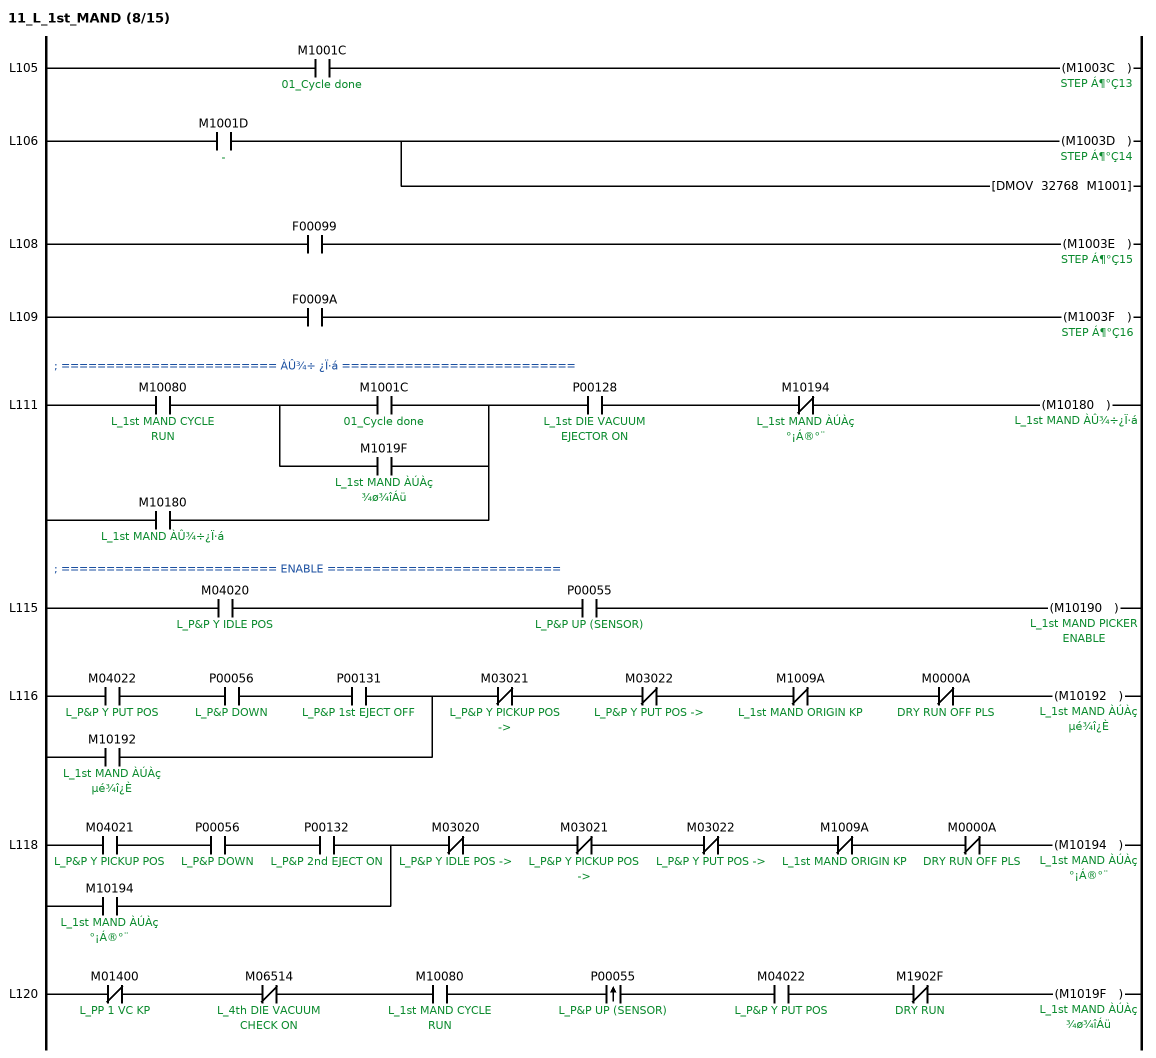
; L105
LOAD      M1001C	// 01_Cycle done
OUT       M1003C	// STEP Á¶°Ç13
; L106
LOAD      M1001D	// -
OUT       M1003D	// STEP Á¶°Ç14
DMOV      32768 M1001
; L108
LOAD      F00099
OUT       M1003E	// STEP Á¶°Ç15
; L109
LOAD      F0009A
OUT       M1003F	// STEP Á¶°Ç16
// ======================== ÀÛ¾÷ ¿Ï·á ==========================
; L111
LOAD      M10080	// L_1st MAND CYCLE RUN
LOAD      M1001C	// 01_Cycle done
OR        M1019F	// L_1st MAND ÀÚÀç ¾ø¾îÁü
AND LOAD
OR        M10180	// L_1st MAND ÀÛ¾÷¿Ï·á
AND       P00128	// L_1st DIE VACUUM EJECTOR ON
AND NOT   M10194	// L_1st MAND ÀÚÀç °¡Á®°¨
OUT       M10180	// L_1st MAND ÀÛ¾÷¿Ï·á
// ======================== ENABLE ==========================
; L115
LOAD      M04020	// L_P&P Y IDLE POS
AND       P00055	// L_P&P UP (SENSOR)
OUT       M10190	// L_1st MAND PICKER ENABLE
; L116
LOAD      M04022	// L_P&P Y PUT POS
AND       P00056	// L_P&P DOWN
AND       P00131	// L_P&P 1st EJECT OFF
OR        M10192	// L_1st MAND ÀÚÀç µé¾î¿È
AND NOT   M03021	// L_P&P Y PICKUP POS ->
AND NOT   M03022	// L_P&P Y PUT POS ->
AND NOT   M1009A	// L_1st MAND ORIGIN KP
AND NOT   M0000A	// DRY RUN OFF PLS
OUT       M10192	// L_1st MAND ÀÚÀç µé¾î¿È
; L118
LOAD      M04021	// L_P&P Y PICKUP POS
AND       P00056	// L_P&P DOWN
AND       P00132	// L_P&P 2nd EJECT ON
OR        M10194	// L_1st MAND ÀÚÀç °¡Á®°¨
AND NOT   M03020	// L_P&P Y IDLE POS ->
AND NOT   M03021	// L_P&P Y PICKUP POS ->
AND NOT   M03022	// L_P&P Y PUT POS ->
AND NOT   M1009A	// L_1st MAND ORIGIN KP
AND NOT   M0000A	// DRY RUN OFF PLS
OUT       M10194	// L_1st MAND ÀÚÀç °¡Á®°¨
; L120
LOAD NOT  M01400	// L_PP 1 VC KP
AND NOT   M06514	// L_4th DIE VACUUM CHECK ON
AND       M10080	// L_1st MAND CYCLE RUN
ANDP      P00055	// L_P&P UP (SENSOR)
AND       M04022	// L_P&P Y PUT POS
AND NOT   M1902F	// DRY RUN
OUT       M1019F	// L_1st MAND ÀÚÀç ¾ø¾îÁü

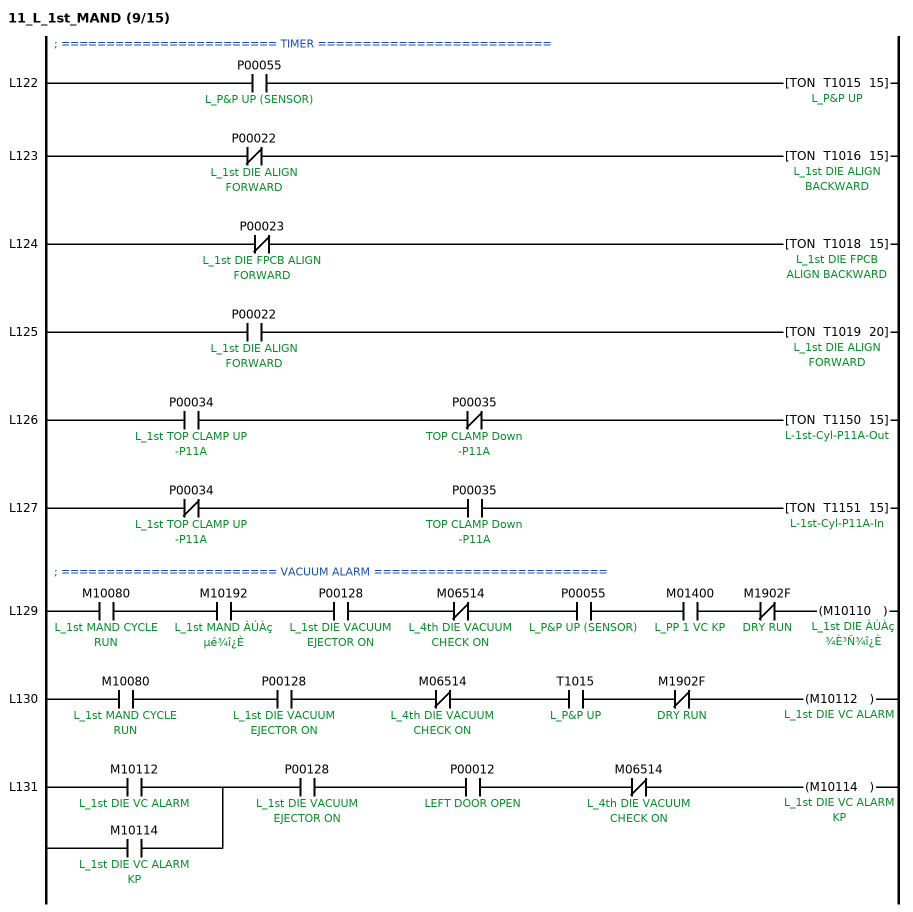
// ======================== TIMER ==========================
; L122
LOAD      P00055	// L_P&P UP (SENSOR)
TON       T1015 15	// L_P&P UP
; L123
LOAD NOT  P00022	// L_1st DIE ALIGN FORWARD
TON       T1016 15	// L_1st DIE ALIGN BACKWARD
; L124
LOAD NOT  P00023	// L_1st DIE FPCB ALIGN FORWARD
TON       T1018 15	// L_1st DIE FPCB ALIGN BACKWARD
; L125
LOAD      P00022	// L_1st DIE ALIGN FORWARD
TON       T1019 20	// L_1st DIE ALIGN FORWARD
; L126
LOAD      P00034	// L_1st TOP CLAMP UP -P11A
AND NOT   P00035	// TOP CLAMP Down -P11A
TON       T1150 15	// L-1st-Cyl-P11A-Out
; L127
LOAD NOT  P00034	// L_1st TOP CLAMP UP -P11A
AND       P00035	// TOP CLAMP Down -P11A
TON       T1151 15	// L-1st-Cyl-P11A-In
// ======================== VACUUM ALARM ==========================
; L129
LOAD      M10080	// L_1st MAND CYCLE RUN
AND       M10192	// L_1st MAND ÀÚÀç µé¾î¿È
AND       P00128	// L_1st DIE VACUUM EJECTOR ON
AND NOT   M06514	// L_4th DIE VACUUM CHECK ON
AND       P00055	// L_P&P UP (SENSOR)
AND       M01400	// L_PP 1 VC KP
AND NOT   M1902F	// DRY RUN
OUT       M10110	// L_1st DIE ÀÚÀç ¾È³Ñ¾î¿È
; L130
LOAD      M10080	// L_1st MAND CYCLE RUN
AND       P00128	// L_1st DIE VACUUM EJECTOR ON
AND NOT   M06514	// L_4th DIE VACUUM CHECK ON
AND       T1015	// L_P&P UP
AND NOT   M1902F	// DRY RUN
OUT       M10112	// L_1st DIE VC ALARM
; L131
LOAD      M10112	// L_1st DIE VC ALARM
OR        M10114	// L_1st DIE VC ALARM KP
AND       P00128	// L_1st DIE VACUUM EJECTOR ON
AND       P00012	// LEFT DOOR OPEN
AND NOT   M06514	// L_4th DIE VACUUM CHECK ON
OUT       M10114	// L_1st DIE VC ALARM KP

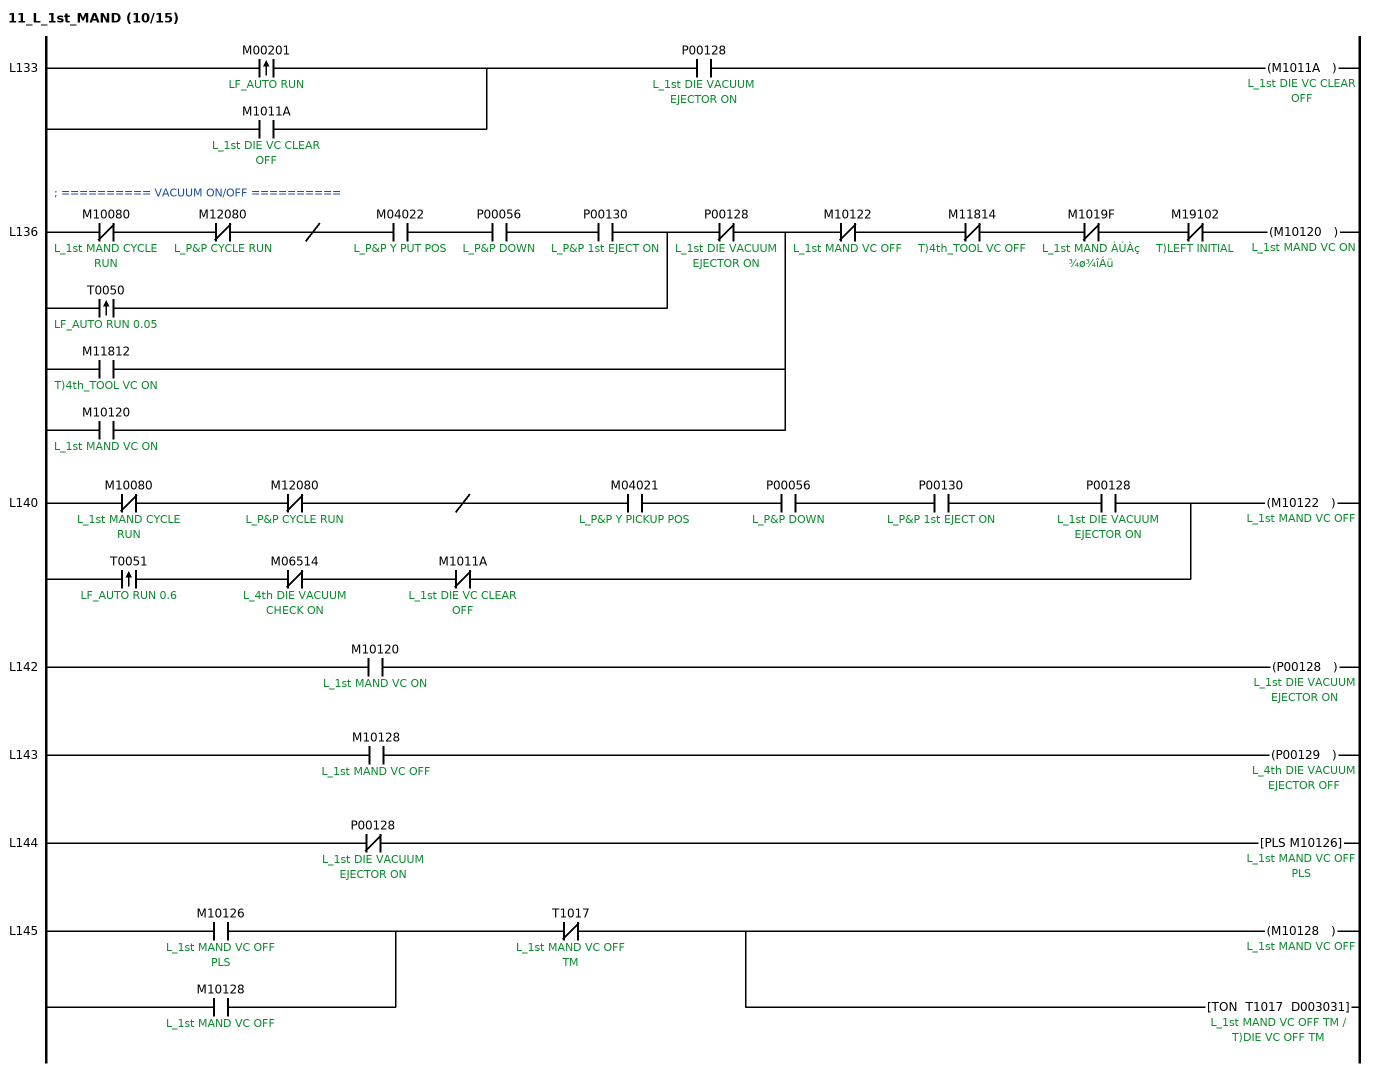
; L133
LOADP     M00201	// LF_AUTO RUN
OR        M1011A	// L_1st DIE VC CLEAR OFF
AND       P00128	// L_1st DIE VACUUM EJECTOR ON
OUT       M1011A	// L_1st DIE VC CLEAR OFF
// ========== VACUUM ON/OFF ==========
; L136
LOAD NOT  M10080	// L_1st MAND CYCLE RUN
AND NOT   M12080	// L_P&P CYCLE RUN
NOT
AND       M04022	// L_P&P Y PUT POS
AND       P00056	// L_P&P DOWN
AND       P00130	// L_P&P 1st EJECT ON
ORP       T0050	// LF_AUTO RUN 0.05
AND NOT   P00128	// L_1st DIE VACUUM EJECTOR ON
OR        M11812	// T)4th_TOOL VC ON
OR        M10120	// L_1st MAND VC ON
AND NOT   M10122	// L_1st MAND VC OFF
AND NOT   M11814	// T)4th_TOOL VC OFF
AND NOT   M1019F	// L_1st MAND ÀÚÀç ¾ø¾îÁü
AND NOT   M19102	// T)LEFT INITIAL
OUT       M10120	// L_1st MAND VC ON
; L140
LOAD NOT  M10080	// L_1st MAND CYCLE RUN
AND NOT   M12080	// L_P&P CYCLE RUN
NOT
AND       M04021	// L_P&P Y PICKUP POS
AND       P00056	// L_P&P DOWN
AND       P00130	// L_P&P 1st EJECT ON
AND       P00128	// L_1st DIE VACUUM EJECTOR ON
LOADP     T0051	// LF_AUTO RUN 0.6
AND NOT   M06514	// L_4th DIE VACUUM CHECK ON
AND NOT   M1011A	// L_1st DIE VC CLEAR OFF
OR LOAD
OUT       M10122	// L_1st MAND VC OFF
; L142
LOAD      M10120	// L_1st MAND VC ON
OUT       P00128	// L_1st DIE VACUUM EJECTOR ON
; L143
LOAD      M10128	// L_1st MAND VC OFF
OUT       P00129	// L_4th DIE VACUUM EJECTOR OFF
; L144
LOAD NOT  P00128	// L_1st DIE VACUUM EJECTOR ON
OUTP      M10126	// L_1st MAND VC OFF PLS
; L145
LOAD      M10126	// L_1st MAND VC OFF PLS
OR        M10128	// L_1st MAND VC OFF
AND NOT   T1017	// L_1st MAND VC OFF TM
OUT       M10128	// L_1st MAND VC OFF
TON       T1017 D003031	// L_1st MAND VC OFF TM / T)DIE VC OFF TM

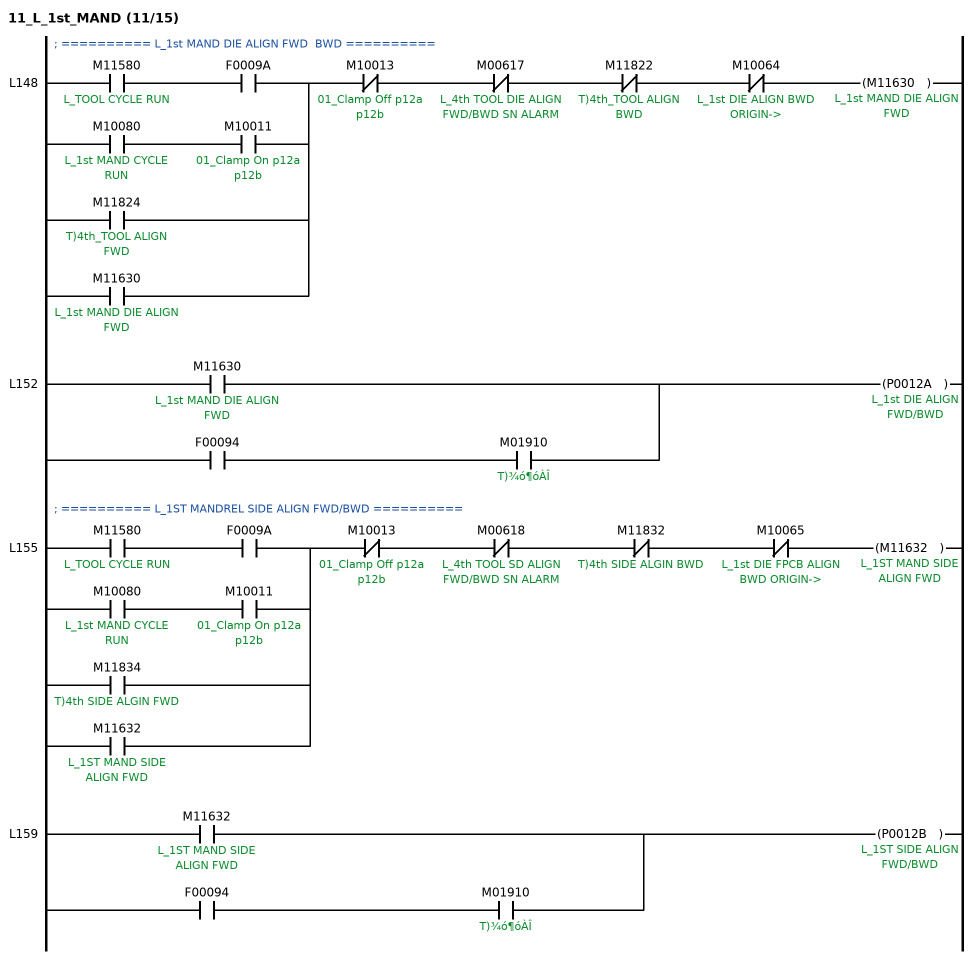
// ========== L_1st MAND DIE ALIGN FWD  BWD ==========
; L148
LOAD      M11580	// L_TOOL CYCLE RUN
AND       F0009A
LOAD      M10080	// L_1st MAND CYCLE RUN
AND       M10011	// 01_Clamp On p12a p12b
OR LOAD
OR        M11824	// T)4th_TOOL ALIGN FWD
OR        M11630	// L_1st MAND DIE ALIGN FWD
AND NOT   M10013	// 01_Clamp Off p12a p12b
AND NOT   M00617	// L_4th TOOL DIE ALIGN FWD/BWD SN ALARM
AND NOT   M11822	// T)4th_TOOL ALIGN BWD
AND NOT   M10064	// L_1st DIE ALIGN BWD ORIGIN->
OUT       M11630	// L_1st MAND DIE ALIGN FWD
; L152
LOAD      M11630	// L_1st MAND DIE ALIGN FWD
LOAD      F00094
AND       M01910	// T)¾ó¶óÀÎ
OR LOAD
OUT       P0012A	// L_1st DIE ALIGN FWD/BWD
// ========== L_1ST MANDREL SIDE ALIGN FWD/BWD ==========
; L155
LOAD      M11580	// L_TOOL CYCLE RUN
AND       F0009A
LOAD      M10080	// L_1st MAND CYCLE RUN
AND       M10011	// 01_Clamp On p12a p12b
OR LOAD
OR        M11834	// T)4th SIDE ALGIN FWD
OR        M11632	// L_1ST MAND SIDE ALIGN FWD
AND NOT   M10013	// 01_Clamp Off p12a p12b
AND NOT   M00618	// L_4th TOOL SD ALIGN FWD/BWD SN ALARM
AND NOT   M11832	// T)4th SIDE ALGIN BWD
AND NOT   M10065	// L_1st DIE FPCB ALIGN BWD ORIGIN->
OUT       M11632	// L_1ST MAND SIDE ALIGN FWD
; L159
LOAD      M11632	// L_1ST MAND SIDE ALIGN FWD
LOAD      F00094
AND       M01910	// T)¾ó¶óÀÎ
OR LOAD
OUT       P0012B	// L_1ST SIDE ALIGN FWD/BWD

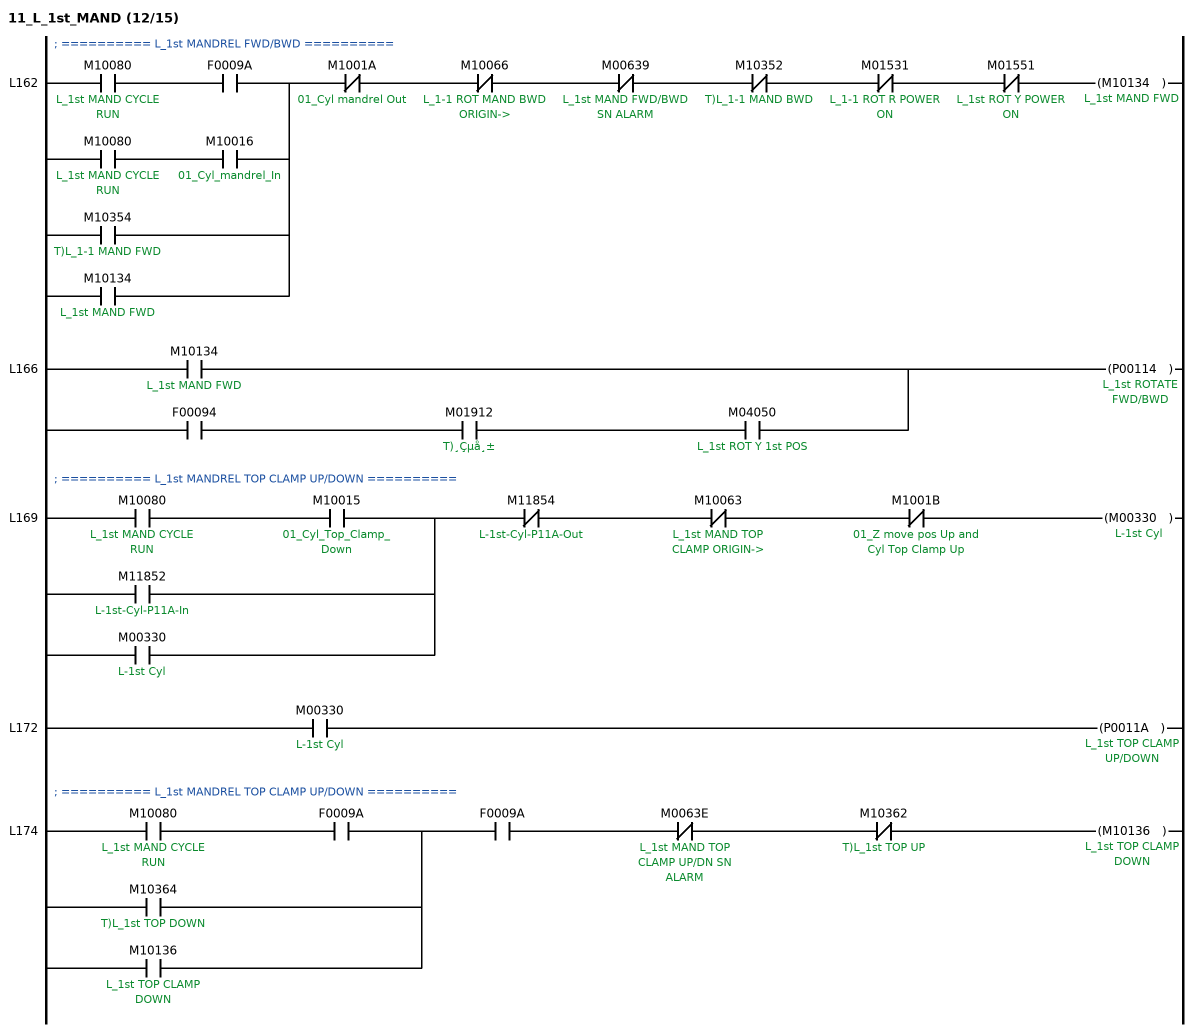
// ========== L_1st MANDREL FWD/BWD ==========
; L162
LOAD      M10080	// L_1st MAND CYCLE RUN
AND       F0009A
LOAD      M10080	// L_1st MAND CYCLE RUN
AND       M10016	// 01_Cyl_mandrel_In
OR LOAD
OR        M10354	// T)L_1-1 MAND FWD
OR        M10134	// L_1st MAND FWD
AND NOT   M1001A	// 01_Cyl mandrel Out
AND NOT   M10066	// L_1-1 ROT MAND BWD ORIGIN->
AND NOT   M00639	// L_1st MAND FWD/BWD SN ALARM
AND NOT   M10352	// T)L_1-1 MAND BWD
AND NOT   M01531	// L_1-1 ROT R POWER ON
AND NOT   M01551	// L_1st ROT Y POWER ON
OUT       M10134	// L_1st MAND FWD
; L166
LOAD      M10134	// L_1st MAND FWD
LOAD      F00094
AND       M01912	// T)¸Çµå¸±
AND       M04050	// L_1st ROT Y 1st POS
OR LOAD
OUT       P00114	// L_1st ROTATE FWD/BWD
// ========== L_1st MANDREL TOP CLAMP UP/DOWN ==========
; L169
LOAD      M10080	// L_1st MAND CYCLE RUN
AND       M10015	// 01_Cyl_Top_Clamp_Down
OR        M11852	// L-1st-Cyl-P11A-In
OR        M00330	// L-1st Cyl
AND NOT   M11854	// L-1st-Cyl-P11A-Out
AND NOT   M10063	// L_1st MAND TOP CLAMP ORIGIN->
AND NOT   M1001B	// 01_Z move pos Up and Cyl Top Clamp Up
OUT       M00330	// L-1st Cyl
; L172
LOAD      M00330	// L-1st Cyl
OUT       P0011A	// L_1st TOP CLAMP UP/DOWN
// ========== L_1st MANDREL TOP CLAMP UP/DOWN ==========
; L174
LOAD      M10080	// L_1st MAND CYCLE RUN
AND       F0009A
OR        M10364	// T)L_1st TOP DOWN
OR        M10136	// L_1st TOP CLAMP DOWN
AND       F0009A
AND NOT   M0063E	// L_1st MAND TOP CLAMP UP/DN SN ALARM
AND NOT   M10362	// T)L_1st TOP UP
OUT       M10136	// L_1st TOP CLAMP DOWN

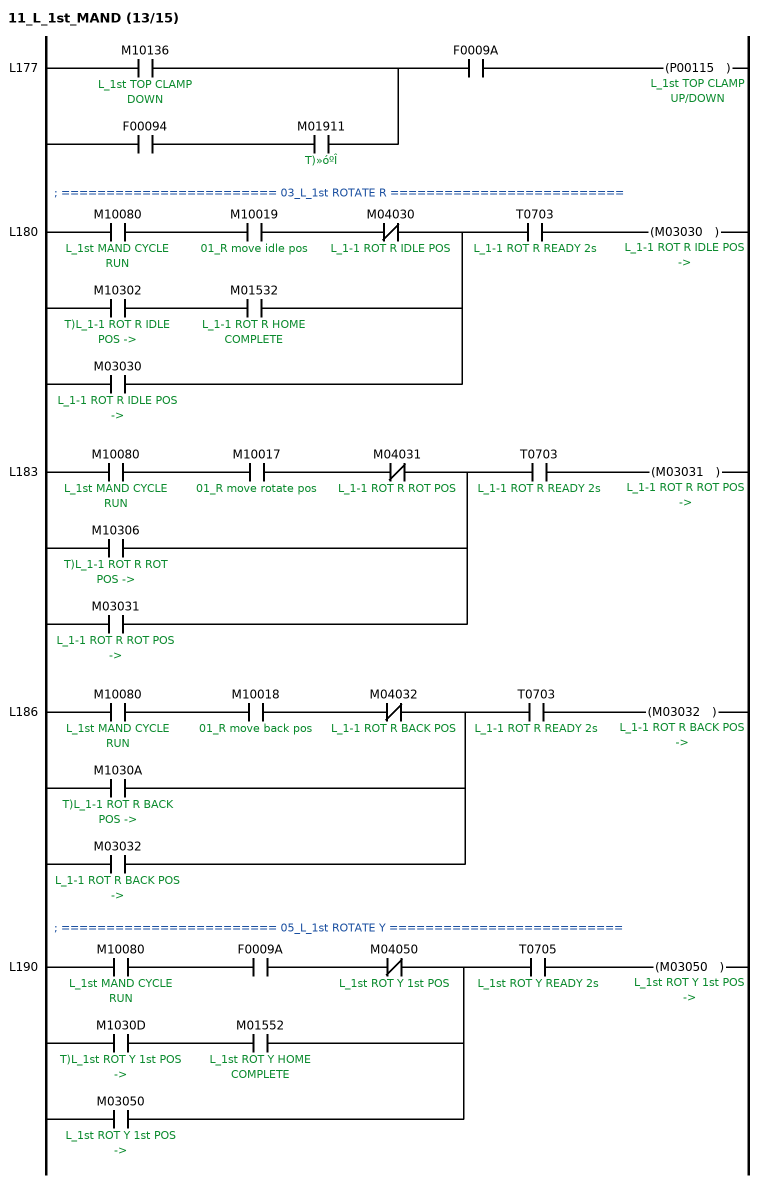
; L177
LOAD      M10136	// L_1st TOP CLAMP DOWN
LOAD      F00094
AND       M01911	// T)»óºÎ
OR LOAD
AND       F0009A
OUT       P00115	// L_1st TOP CLAMP UP/DOWN
// ======================== 03_L_1st ROTATE R ==========================
; L180
LOAD      M10080	// L_1st MAND CYCLE RUN
AND       M10019	// 01_R move idle pos
AND NOT   M04030	// L_1-1 ROT R IDLE POS
LOAD      M10302	// T)L_1-1 ROT R IDLE POS ->
AND       M01532	// L_1-1 ROT R HOME COMPLETE
OR LOAD
OR        M03030	// L_1-1 ROT R IDLE POS ->
AND       T0703	// L_1-1 ROT R READY 2s
OUT       M03030	// L_1-1 ROT R IDLE POS ->
; L183
LOAD      M10080	// L_1st MAND CYCLE RUN
AND       M10017	// 01_R move rotate pos
AND NOT   M04031	// L_1-1 ROT R ROT POS
OR        M10306	// T)L_1-1 ROT R ROT POS ->
OR        M03031	// L_1-1 ROT R ROT POS ->
AND       T0703	// L_1-1 ROT R READY 2s
OUT       M03031	// L_1-1 ROT R ROT POS ->
; L186
LOAD      M10080	// L_1st MAND CYCLE RUN
AND       M10018	// 01_R move back pos
AND NOT   M04032	// L_1-1 ROT R BACK POS
OR        M1030A	// T)L_1-1 ROT R BACK POS ->
OR        M03032	// L_1-1 ROT R BACK POS ->
AND       T0703	// L_1-1 ROT R READY 2s
OUT       M03032	// L_1-1 ROT R BACK POS ->
// ======================== 05_L_1st ROTATE Y ==========================
; L190
LOAD      M10080	// L_1st MAND CYCLE RUN
AND       F0009A
AND NOT   M04050	// L_1st ROT Y 1st POS
LOAD      M1030D	// T)L_1st ROT Y 1st POS ->
AND       M01552	// L_1st ROT Y HOME COMPLETE
OR LOAD
OR        M03050	// L_1st ROT Y 1st POS ->
AND       T0705	// L_1st ROT Y READY 2s
OUT       M03050	// L_1st ROT Y 1st POS ->

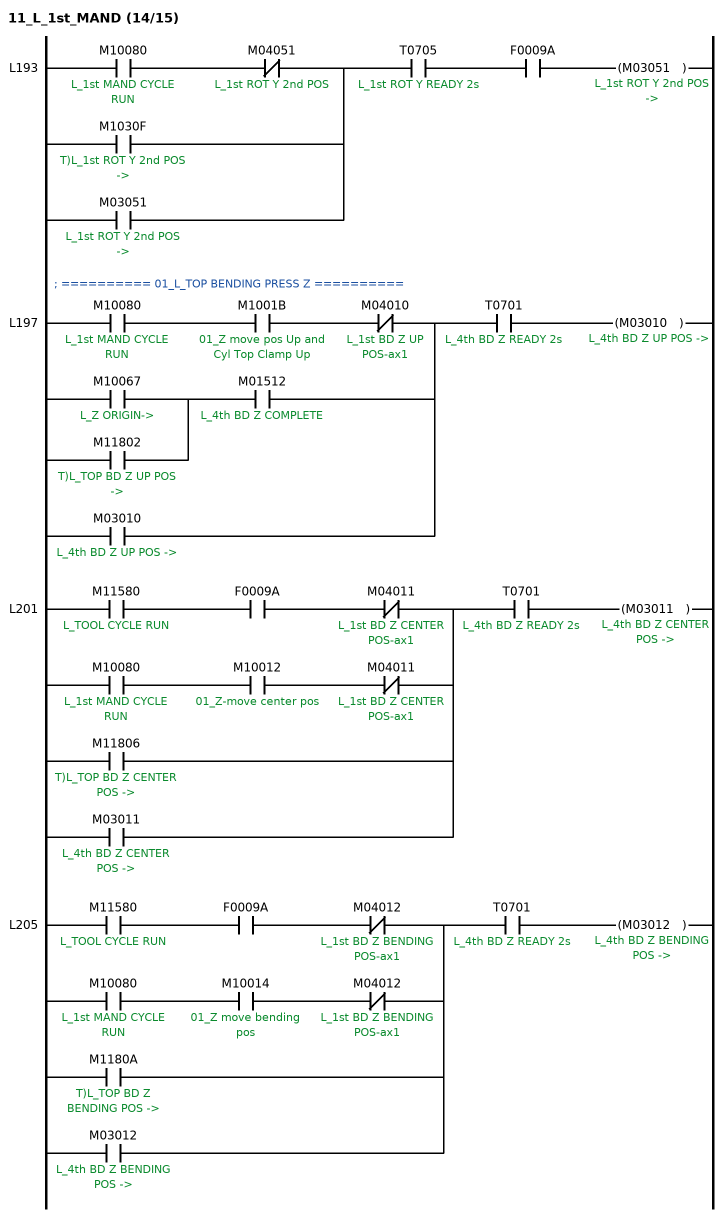
; L193
LOAD      M10080	// L_1st MAND CYCLE RUN
AND NOT   M04051	// L_1st ROT Y 2nd POS
OR        M1030F	// T)L_1st ROT Y 2nd POS ->
OR        M03051	// L_1st ROT Y 2nd POS ->
AND       T0705	// L_1st ROT Y READY 2s
AND       F0009A
OUT       M03051	// L_1st ROT Y 2nd POS ->
// ========== 01_L_TOP BENDING PRESS Z ==========
; L197
LOAD      M10080	// L_1st MAND CYCLE RUN
AND       M1001B	// 01_Z move pos Up and Cyl Top Clamp Up
AND NOT   M04010	// L_1st BD Z UP POS-ax1
LOAD      M10067	// L_Z ORIGIN->
OR        M11802	// T)L_TOP BD Z UP POS ->
AND       M01512	// L_4th BD Z COMPLETE
OR LOAD
OR        M03010	// L_4th BD Z UP POS ->
AND       T0701	// L_4th BD Z READY 2s
OUT       M03010	// L_4th BD Z UP POS ->
; L201
LOAD      M11580	// L_TOOL CYCLE RUN
AND       F0009A
AND NOT   M04011	// L_1st BD Z CENTER POS-ax1
LOAD      M10080	// L_1st MAND CYCLE RUN
AND       M10012	// 01_Z-move center pos
AND NOT   M04011	// L_1st BD Z CENTER POS-ax1
OR LOAD
OR        M11806	// T)L_TOP BD Z CENTER POS ->
OR        M03011	// L_4th BD Z CENTER POS ->
AND       T0701	// L_4th BD Z READY 2s
OUT       M03011	// L_4th BD Z CENTER POS ->
; L205
LOAD      M11580	// L_TOOL CYCLE RUN
AND       F0009A
AND NOT   M04012	// L_1st BD Z BENDING POS-ax1
LOAD      M10080	// L_1st MAND CYCLE RUN
AND       M10014	// 01_Z move bending pos
AND NOT   M04012	// L_1st BD Z BENDING POS-ax1
OR LOAD
OR        M1180A	// T)L_TOP BD Z BENDING POS ->
OR        M03012	// L_4th BD Z BENDING POS ->
AND       T0701	// L_4th BD Z READY 2s
OUT       M03012	// L_4th BD Z BENDING POS ->

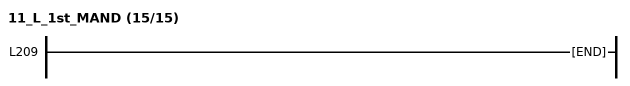
; L209
END

PROGRAM 12_L_2nd_MAND (task: ½ºÄµ ÇÁ·Î±×·¥)

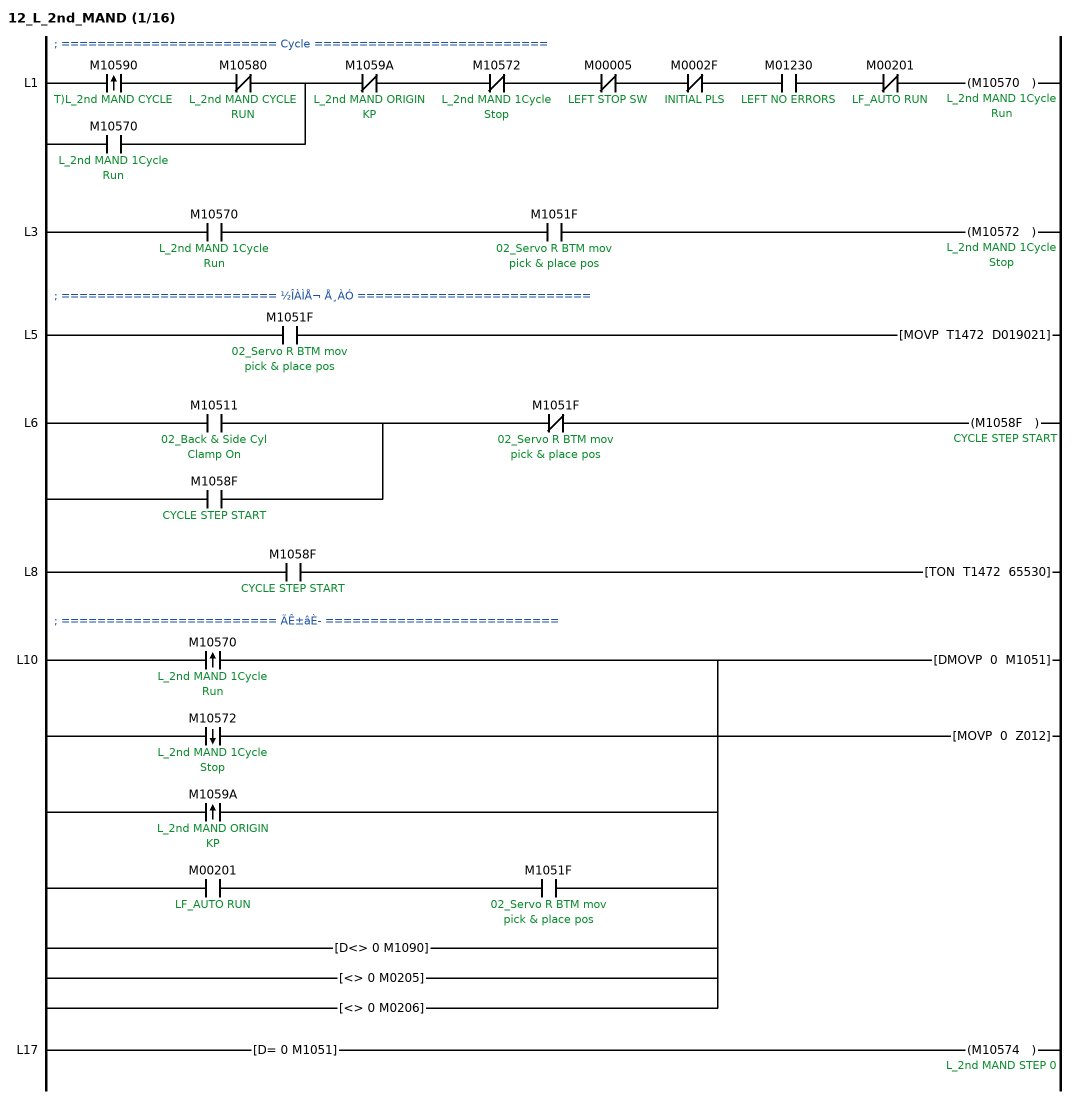
// ======================== Cycle ==========================
; L1
LOADP     M10590	// T)L_2nd MAND CYCLE
AND NOT   M10580	// L_2nd MAND CYCLE RUN
OR        M10570	// L_2nd MAND 1Cycle Run
AND NOT   M1059A	// L_2nd MAND ORIGIN KP
AND NOT   M10572	// L_2nd MAND 1Cycle Stop
AND NOT   M00005	// LEFT STOP SW
AND NOT   M0002F	// INITIAL PLS
AND       M01230	// LEFT NO ERRORS
AND NOT   M00201	// LF_AUTO RUN
OUT       M10570	// L_2nd MAND 1Cycle Run
; L3
LOAD      M10570	// L_2nd MAND 1Cycle Run
AND       M1051F	// 02_Servo R BTM mov pick & place pos
OUT       M10572	// L_2nd MAND 1Cycle Stop
// ======================== ½ÎÀÌÅ¬ Å¸ÀÓ ==========================
; L5
LOAD      M1051F	// 02_Servo R BTM mov pick & place pos
MOVP      T1472 D019021
; L6
LOAD      M10511	// 02_Back & Side Cyl Clamp On
OR        M1058F	// CYCLE STEP START
AND NOT   M1051F	// 02_Servo R BTM mov pick & place pos
OUT       M1058F	// CYCLE STEP START
; L8
LOAD      M1058F	// CYCLE STEP START
TON       T1472 65530
// ======================== ÃÊ±âÈ­ ==========================
; L10
LOADP     M10570	// L_2nd MAND 1Cycle Run
ORN       M10572	// L_2nd MAND 1Cycle Stop
ORP       M1059A	// L_2nd MAND ORIGIN KP
LOAD      M00201	// LF_AUTO RUN
AND       M1051F	// 02_Servo R BTM mov pick & place pos
OR LOAD
ORD<>     0 M1090
OR<>      0 M0205
OR<>      0 M0206
DMOVP     0 M1051
MOVP      0 Z012
; L17
LOADD=    0 M1051
OUT       M10574	// L_2nd MAND STEP 0

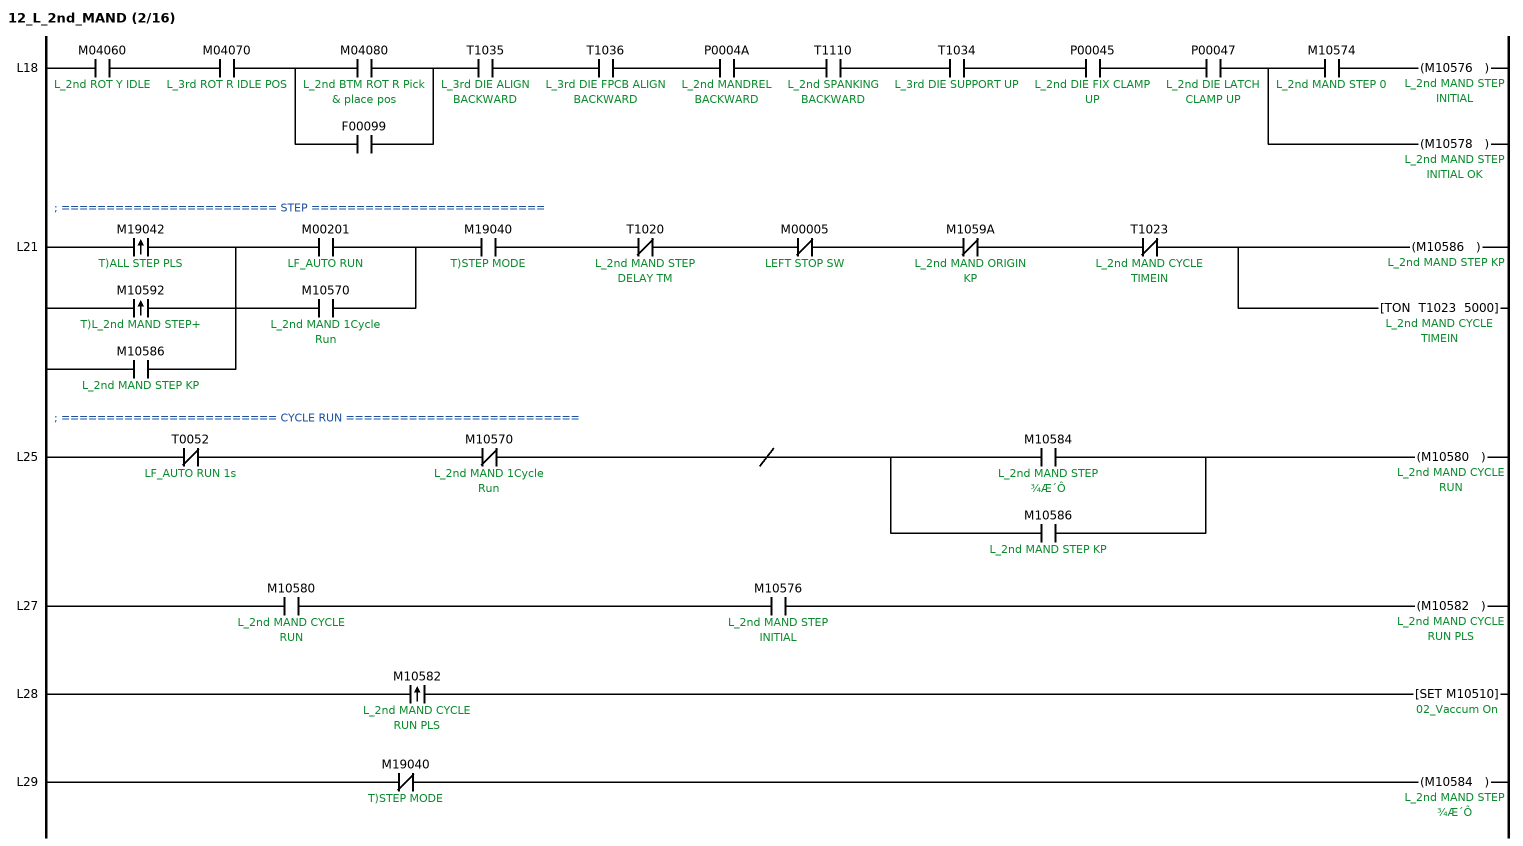
; L18
LOAD      M04060	// L_2nd ROT Y IDLE
AND       M04070	// L_3rd ROT R IDLE POS
LOAD      M04080	// L_2nd BTM ROT R Pick & place pos
OR        F00099
AND LOAD
AND       T1035	// L_3rd DIE ALIGN BACKWARD
AND       T1036	// L_3rd DIE FPCB ALIGN BACKWARD
AND       P0004A	// L_2nd MANDREL BACKWARD
AND       T1110	// L_2nd SPANKING BACKWARD
AND       T1034	// L_3rd DIE SUPPORT UP
AND       P00045	// L_2nd DIE FIX CLAMP UP
AND       P00047	// L_2nd DIE LATCH CLAMP UP
MPUSH
AND       M10574	// L_2nd MAND STEP 0
OUT       M10576	// L_2nd MAND STEP INITIAL
MPOP
OUT       M10578	// L_2nd MAND STEP INITIAL OK
// ======================== STEP ==========================
; L21
LOADP     M19042	// T)ALL STEP PLS
ORP       M10592	// T)L_2nd MAND STEP+
OR        M10586	// L_2nd MAND STEP KP
LOAD      M00201	// LF_AUTO RUN
OR        M10570	// L_2nd MAND 1Cycle Run
AND LOAD
AND       M19040	// T)STEP MODE
AND NOT   T1020	// L_2nd MAND STEP DELAY TM
AND NOT   M00005	// LEFT STOP SW
AND NOT   M1059A	// L_2nd MAND ORIGIN KP
AND NOT   T1023	// L_2nd MAND CYCLE TIMEIN
OUT       M10586	// L_2nd MAND STEP KP
TON       T1023 5000	// L_2nd MAND CYCLE TIMEIN
// ======================== CYCLE RUN ==========================
; L25
LOAD NOT  T0052	// LF_AUTO RUN 1s
AND NOT   M10570	// L_2nd MAND 1Cycle Run
NOT
LOAD      M10584	// L_2nd MAND STEP ¾Æ´Ô
OR        M10586	// L_2nd MAND STEP KP
AND LOAD
OUT       M10580	// L_2nd MAND CYCLE RUN
; L27
LOAD      M10580	// L_2nd MAND CYCLE RUN
AND       M10576	// L_2nd MAND STEP INITIAL
OUT       M10582	// L_2nd MAND CYCLE RUN PLS
; L28
LOADP     M10582	// L_2nd MAND CYCLE RUN PLS
SET       M10510	// 02_Vaccum On
; L29
LOAD NOT  M19040	// T)STEP MODE
OUT       M10584	// L_2nd MAND STEP ¾Æ´Ô

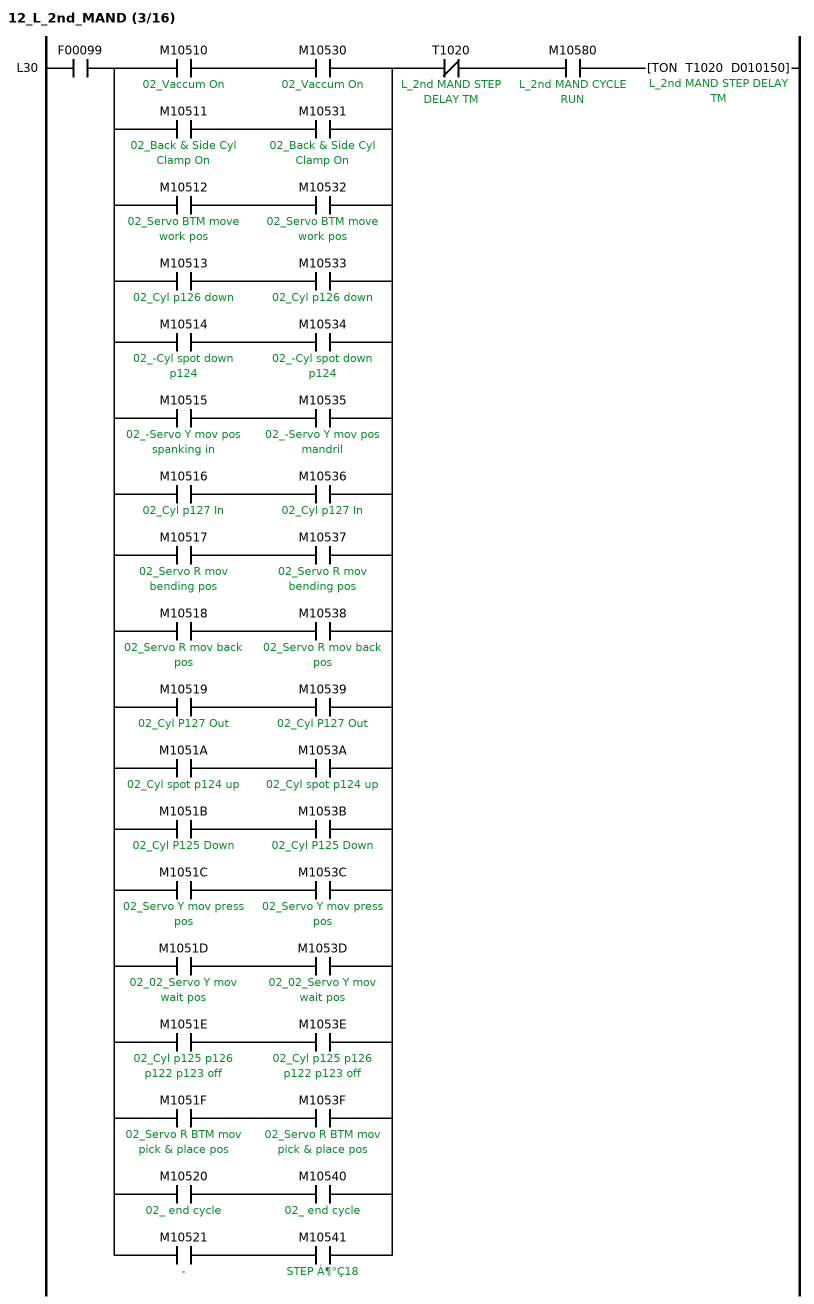
; L30
LOAD      F00099
LOAD      M10510	// 02_Vaccum On
AND       M10530	// 02_Vaccum On
LOAD      M10511	// 02_Back & Side Cyl Clamp On
AND       M10531	// 02_Back & Side Cyl Clamp On
OR LOAD
LOAD      M10512	// 02_Servo BTM move work pos
AND       M10532	// 02_Servo BTM move work pos
OR LOAD
LOAD      M10513	// 02_Cyl p126 down
AND       M10533	// 02_Cyl p126 down
OR LOAD
LOAD      M10514	// 02_-Cyl spot down p124
AND       M10534	// 02_-Cyl spot down p124
OR LOAD
LOAD      M10515	// 02_-Servo Y mov pos spanking in
AND       M10535	// 02_-Servo Y mov pos mandril
OR LOAD
LOAD      M10516	// 02_Cyl p127 In
AND       M10536	// 02_Cyl p127 In
OR LOAD
LOAD      M10517	// 02_Servo R mov bending pos
AND       M10537	// 02_Servo R mov bending pos
OR LOAD
LOAD      M10518	// 02_Servo R mov back pos
AND       M10538	// 02_Servo R mov back pos
OR LOAD
LOAD      M10519	// 02_Cyl P127 Out
AND       M10539	// 02_Cyl P127 Out
OR LOAD
LOAD      M1051A	// 02_Cyl spot p124 up
AND       M1053A	// 02_Cyl spot p124 up
OR LOAD
LOAD      M1051B	// 02_Cyl P125 Down
AND       M1053B	// 02_Cyl P125 Down
OR LOAD
LOAD      M1051C	// 02_Servo Y mov press pos
AND       M1053C	// 02_Servo Y mov press pos
OR LOAD
LOAD      M1051D	// 02_02_Servo Y mov wait pos
AND       M1053D	// 02_02_Servo Y mov wait pos
OR LOAD
LOAD      M1051E	// 02_Cyl p125 p126 p122 p123 off
AND       M1053E	// 02_Cyl p125 p126 p122 p123 off
OR LOAD
LOAD      M1051F	// 02_Servo R BTM mov pick & place pos
AND       M1053F	// 02_Servo R BTM mov pick & place pos
OR LOAD
LOAD      M10520	// 02_ end cycle
AND       M10540	// 02_ end cycle
OR LOAD
LOAD      M10521	// -
AND       M10541	// STEP Á¶°Ç18
OR LOAD
AND LOAD
AND NOT   T1020	// L_2nd MAND STEP DELAY TM
AND       M10580	// L_2nd MAND CYCLE RUN
TON       T1020 D010150	// L_2nd MAND STEP DELAY TM

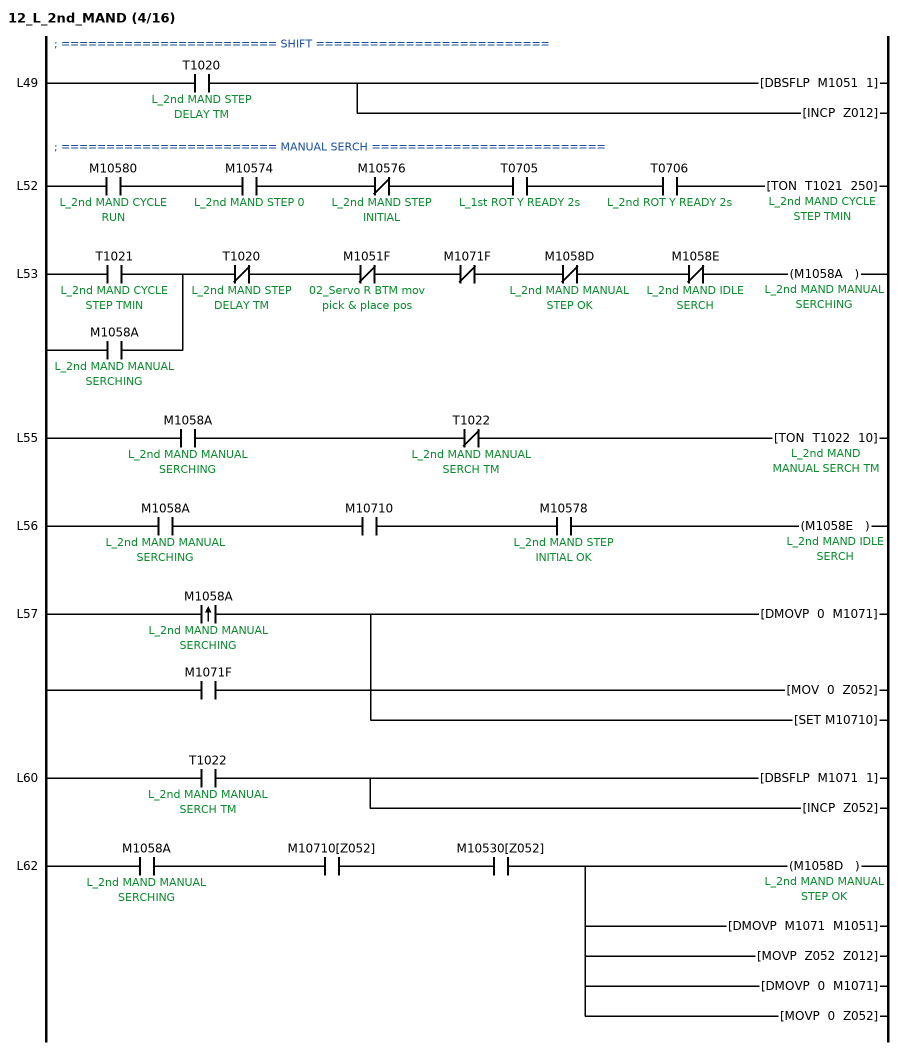
// ======================== SHIFT ==========================
; L49
LOAD      T1020	// L_2nd MAND STEP DELAY TM
DBSFLP    M1051 1
INCP      Z012
// ======================== MANUAL SERCH ==========================
; L52
LOAD      M10580	// L_2nd MAND CYCLE RUN
AND       M10574	// L_2nd MAND STEP 0
AND NOT   M10576	// L_2nd MAND STEP INITIAL
AND       T0705	// L_1st ROT Y READY 2s
AND       T0706	// L_2nd ROT Y READY 2s
TON       T1021 250	// L_2nd MAND CYCLE STEP TMIN
; L53
LOAD      T1021	// L_2nd MAND CYCLE STEP TMIN
OR        M1058A	// L_2nd MAND MANUAL SERCHING
AND NOT   T1020	// L_2nd MAND STEP DELAY TM
AND NOT   M1051F	// 02_Servo R BTM mov pick & place pos
AND NOT   M1071F
AND NOT   M1058D	// L_2nd MAND MANUAL STEP OK
AND NOT   M1058E	// L_2nd MAND IDLE SERCH
OUT       M1058A	// L_2nd MAND MANUAL SERCHING
; L55
LOAD      M1058A	// L_2nd MAND MANUAL SERCHING
AND NOT   T1022	// L_2nd MAND MANUAL SERCH TM
TON       T1022 10	// L_2nd MAND MANUAL SERCH TM
; L56
LOAD      M1058A	// L_2nd MAND MANUAL SERCHING
AND       M10710
AND       M10578	// L_2nd MAND STEP INITIAL OK
OUT       M1058E	// L_2nd MAND IDLE SERCH
; L57
LOADP     M1058A	// L_2nd MAND MANUAL SERCHING
OR        M1071F
DMOVP     0 M1071
MOV       0 Z052
SET       M10710
; L60
LOAD      T1022	// L_2nd MAND MANUAL SERCH TM
DBSFLP    M1071 1
INCP      Z052
; L62
LOAD      M1058A	// L_2nd MAND MANUAL SERCHING
AND       M10710[Z052]
AND       M10530[Z052]
OUT       M1058D	// L_2nd MAND MANUAL STEP OK
DMOVP     M1071 M1051
MOVP      Z052 Z012
DMOVP     0 M1071
MOVP      0 Z052

